//     PlcTask Inputs/MAIN.force_rb_Y[62] <-> Status process data mapping/force_rb_Y
//     PlcTask Inputs/MAIN.force_rb_Z[62] <-> Status process data mapping/force_rb_Z
//     PlcTask Inputs/MAIN.force_sp_X[62] <-> Status process data mapping/force_sp_X
//     PlcTask Inputs/MAIN.force_sp_Y[62] <-> Status process data mapping/force_sp_Y
//     PlcTask Inputs/MAIN.force_sp_Z[62] <-> Status process data mapping/force_sp_Z
//     PlcTask Inputs/MAIN.pwm1[62] <-> Status process data mapping/pwm1
//     PlcTask Inputs/MAIN.pwm2[62] <-> Status process data mapping/pwm2
//     PlcTask Inputs/MAIN.pwm3[62] <-> Status process data mapping/pwm3
//     PlcTask Outputs/MAIN.enable_cmd[62] <-> Control process data mapping/enable
//     PlcTask Outputs/MAIN.force_cmd_X[62] <-> Control process data mapping/force_sp_X
//     PlcTask Outputs/MAIN.force_cmd_Y[62] <-> Control process data mapping/force_sp_Y
//     PlcTask Outputs/MAIN.force_cmd_Z[62] <-> Control process data mapping/force_sp_Z
//     PlcTask Outputs/MAIN.msthb[67] <-> Control process data mapping/msthb
//   SAsetGains/SAsetGains Instance <-> Device 1 (EtherCAT)/Box 63 (m1eph)/Box 68 (m1sa)
//     PlcTask Inputs/MAIN.cloop_stat[63] <-> Status process data mapping/close_loop
//     PlcTask Inputs/MAIN.enable_stat[63] <-> Status process data mapping/enable
//     PlcTask Inputs/MAIN.force_rb_X[63] <-> Status process data mapping/force_rb_X
//     PlcTask Inputs/MAIN.force_rb_Y[63] <-> Status process data mapping/force_rb_Y
//     PlcTask Inputs/MAIN.force_rb_Z[63] <-> Status process data mapping/force_rb_Z
//     PlcTask Inputs/MAIN.force_sp_X[63] <-> Status process data mapping/force_sp_X
//     PlcTask Inputs/MAIN.force_sp_Y[63] <-> Status process data mapping/force_sp_Y
//     PlcTask Inputs/MAIN.force_sp_Z[63] <-> Status process data mapping/force_sp_Z
//     PlcTask Inputs/MAIN.pwm1[63] <-> Status process data mapping/pwm1
//     PlcTask Inputs/MAIN.pwm2[63] <-> Status process data mapping/pwm2
//     PlcTask Inputs/MAIN.pwm3[63] <-> Status process data mapping/pwm3
//     PlcTask Outputs/MAIN.enable_cmd[63] <-> Control process data mapping/enable
//     PlcTask Outputs/MAIN.force_cmd_X[63] <-> Control process data mapping/force_sp_X
//     PlcTask Outputs/MAIN.force_cmd_Y[63] <-> Control process data mapping/force_sp_Y
//     PlcTask Outputs/MAIN.force_cmd_Z[63] <-> Control process data mapping/force_sp_Z
//     PlcTask Outputs/MAIN.msthb[68] <-> Control process data mapping/msthb
//   SAsetGains/SAsetGains Instance <-> Device 1 (EtherCAT)/Box 63 (m1eph)/Box 69 (m1sa)
//     PlcTask Inputs/MAIN.cloop_stat[64] <-> Status process data mapping/close_loop
//     PlcTask Inputs/MAIN.enable_stat[64] <-> Status process data mapping/enable
//     PlcTask Inputs/MAIN.force_rb_X[64] <-> Status process data mapping/force_rb_X
//     PlcTask Inputs/MAIN.force_rb_Y[64] <-> Status process data mapping/force_rb_Y
//     PlcTask Inputs/MAIN.force_rb_Z[64] <-> Status process data mapping/force_rb_Z
//     PlcTask Inputs/MAIN.force_sp_X[64] <-> Status process data mapping/force_sp_X
//     PlcTask Inputs/MAIN.force_sp_Y[64] <-> Status process data mapping/force_sp_Y
//     PlcTask Inputs/MAIN.force_sp_Z[64] <-> Status process data mapping/force_sp_Z
//     PlcTask Inputs/MAIN.pwm1[64] <-> Status process data mapping/pwm1
//     PlcTask Inputs/MAIN.pwm2[64] <-> Status process data mapping/pwm2
//     PlcTask Inputs/MAIN.pwm3[64] <-> Status process data mapping/pwm3
//     PlcTask Outputs/MAIN.enable_cmd[64] <-> Control process data mapping/enable
//     PlcTask Outputs/MAIN.force_cmd_X[64] <-> Control process data mapping/force_sp_X
//     PlcTask Outputs/MAIN.force_cmd_Y[64] <-> Control process data mapping/force_sp_Y
//     PlcTask Outputs/MAIN.force_cmd_Z[64] <-> Control process data mapping/force_sp_Z
//     PlcTask Outputs/MAIN.msthb[69] <-> Control process data mapping/msthb
//   SAsetGains/SAsetGains Instance <-> Device 1 (EtherCAT)/Box 63 (m1eph)/Box 70 (m1sa)
//     PlcTask Inputs/MAIN.cloop_stat[65] <-> Status process data mapping/close_loop
//     PlcTask Inputs/MAIN.enable_stat[65] <-> Status process data mapping/enable
//     PlcTask Inputs/MAIN.force_rb_X[65] <-> Status process data mapping/force_rb_X
//     PlcTask Inputs/MAIN.force_rb_Y[65] <-> Status process data mapping/force_rb_Y
//     PlcTask Inputs/MAIN.force_rb_Z[65] <-> Status process data mapping/force_rb_Z
//     PlcTask Inputs/MAIN.force_sp_X[65] <-> Status process data mapping/force_sp_X
//     PlcTask Inputs/MAIN.force_sp_Y[65] <-> Status process data mapping/force_sp_Y
//     PlcTask Inputs/MAIN.force_sp_Z[65] <-> Status process data mapping/force_sp_Z
//     PlcTask Inputs/MAIN.pwm1[65] <-> Status process data mapping/pwm1
//     PlcTask Inputs/MAIN.pwm2[65] <-> Status process data mapping/pwm2
//     PlcTask Inputs/MAIN.pwm3[65] <-> Status process data mapping/pwm3
//     PlcTask Outputs/MAIN.enable_cmd[65] <-> Control process data mapping/enable
//     PlcTask Outputs/MAIN.force_cmd_X[65] <-> Control process data mapping/force_sp_X
//     PlcTask Outputs/MAIN.force_cmd_Y[65] <-> Control process data mapping/force_sp_Y
//     PlcTask Outputs/MAIN.force_cmd_Z[65] <-> Control process data mapping/force_sp_Z
//     PlcTask Outputs/MAIN.msthb[70] <-> Control process data mapping/msthb
//   SAsetGains/SAsetGains Instance <-> Device 1 (EtherCAT)/Box 63 (m1eph)/Box 71 (m1sa)
//     PlcTask Inputs/MAIN.cloop_stat[66] <-> Status process data mapping/close_loop
//     PlcTask Inputs/MAIN.enable_stat[66] <-> Status process data mapping/enable
//     PlcTask Inputs/MAIN.force_rb_X[66] <-> Status process data mapping/force_rb_X
//     PlcTask Inputs/MAIN.force_rb_Y[66] <-> Status process data mapping/force_rb_Y
//     PlcTask Inputs/MAIN.force_rb_Z[66] <-> Status process data mapping/force_rb_Z
//     PlcTask Inputs/MAIN.force_sp_X[66] <-> Status process data mapping/force_sp_X
//     PlcTask Inputs/MAIN.force_sp_Y[66] <-> Status process data mapping/force_sp_Y
//     PlcTask Inputs/MAIN.force_sp_Z[66] <-> Status process data mapping/force_sp_Z
//     PlcTask Inputs/MAIN.pwm1[66] <-> Status process data mapping/pwm1
//     PlcTask Inputs/MAIN.pwm2[66] <-> Status process data mapping/pwm2
//     PlcTask Inputs/MAIN.pwm3[66] <-> Status process data mapping/pwm3
//     PlcTask Outputs/MAIN.enable_cmd[66] <-> Control process data mapping/enable
//     PlcTask Outputs/MAIN.force_cmd_X[66] <-> Control process data mapping/force_sp_X
//     PlcTask Outputs/MAIN.force_cmd_Y[66] <-> Control process data mapping/force_sp_Y
//     PlcTask Outputs/MAIN.force_cmd_Z[66] <-> Control process data mapping/force_sp_Z
//     PlcTask Outputs/MAIN.msthb[71] <-> Control process data mapping/msthb
//   SAsetGains/SAsetGains Instance <-> Device 1 (EtherCAT)/Box 63 (m1eph)/Box 72 (m1sa)
//     PlcTask Inputs/MAIN.cloop_stat[67] <-> Status process data mapping/close_loop
//     PlcTask Inputs/MAIN.enable_stat[67] <-> Status process data mapping/enable
//     PlcTask Inputs/MAIN.force_rb_X[67] <-> Status process data mapping/force_rb_X
//     PlcTask Inputs/MAIN.force_rb_Y[67] <-> Status process data mapping/force_rb_Y
//     PlcTask Inputs/MAIN.force_rb_Z[67] <-> Status process data mapping/force_rb_Z
//     PlcTask Inputs/MAIN.force_sp_X[67] <-> Status process data mapping/force_sp_X
//     PlcTask Inputs/MAIN.force_sp_Y[67] <-> Status process data mapping/force_sp_Y
//     PlcTask Inputs/MAIN.force_sp_Z[67] <-> Status process data mapping/force_sp_Z
//     PlcTask Inputs/MAIN.pwm1[67] <-> Status process data mapping/pwm1
//     PlcTask Inputs/MAIN.pwm2[67] <-> Status process data mapping/pwm2
//     PlcTask Inputs/MAIN.pwm3[67] <-> Status process data mapping/pwm3
//     PlcTask Outputs/MAIN.enable_cmd[67] <-> Control process data mapping/enable
//     PlcTask Outputs/MAIN.force_cmd_X[67] <-> Control process data mapping/force_sp_X
//     PlcTask Outputs/MAIN.force_cmd_Y[67] <-> Control process data mapping/force_sp_Y
//     PlcTask Outputs/MAIN.force_cmd_Z[67] <-> Control process data mapping/force_sp_Z
//     PlcTask Outputs/MAIN.msthb[72] <-> Control process data mapping/msthb
//   SAsetGains/SAsetGains Instance <-> Device 1 (EtherCAT)/Box 63 (m1eph)/Box 73 (m1sa)
//     PlcTask Inputs/MAIN.cloop_stat[68] <-> Status process data mapping/close_loop
//     PlcTask Inputs/MAIN.enable_stat[68] <-> Status process data mapping/enable
//     PlcTask Inputs/MAIN.force_rb_X[68] <-> Status process data mapping/force_rb_X
//     PlcTask Inputs/MAIN.force_rb_Y[68] <-> Status process data mapping/force_rb_Y
//     PlcTask Inputs/MAIN.force_rb_Z[68] <-> Status process data mapping/force_rb_Z
//     PlcTask Inputs/MAIN.force_sp_X[68] <-> Status process data mapping/force_sp_X
//     PlcTask Inputs/MAIN.force_sp_Y[68] <-> Status process data mapping/force_sp_Y
//     PlcTask Inputs/MAIN.force_sp_Z[68] <-> Status process data mapping/force_sp_Z
//     PlcTask Inputs/MAIN.pwm1[68] <-> Status process data mapping/pwm1
//     PlcTask Inputs/MAIN.pwm2[68] <-> Status process data mapping/pwm2
//     PlcTask Inputs/MAIN.pwm3[68] <-> Status process data mapping/pwm3
//     PlcTask Outputs/MAIN.enable_cmd[68] <-> Control process data mapping/enable
//     PlcTask Outputs/MAIN.force_cmd_X[68] <-> Control process data mapping/force_sp_X
//     PlcTask Outputs/MAIN.force_cmd_Y[68] <-> Control process data mapping/force_sp_Y
//     PlcTask Outputs/MAIN.force_cmd_Z[68] <-> Control process data mapping/force_sp_Z
//     PlcTask Outputs/MAIN.msthb[73] <-> Control process data mapping/msthb
//   SAsetGains/SAsetGains Instance <-> Device 1 (EtherCAT)/Box 63 (m1eph)/Box 74 (m1sa)
//     PlcTask Inputs/MAIN.cloop_stat[69] <-> Status process data mapping/close_loop
//     PlcTask Inputs/MAIN.enable_stat[69] <-> Status process data mapping/enable
//     PlcTask Inputs/MAIN.force_rb_X[69] <-> Status process data mapping/force_rb_X
//     PlcTask Inputs/MAIN.force_rb_Y[69] <-> Status process data mapping/force_rb_Y
//     PlcTask Inputs/MAIN.force_rb_Z[69] <-> Status process data mapping/force_rb_Z
//     PlcTask Inputs/MAIN.force_sp_X[69] <-> Status process data mapping/force_sp_X
//     PlcTask Inputs/MAIN.force_sp_Y[69] <-> Status process data mapping/force_sp_Y
//     PlcTask Inputs/MAIN.force_sp_Z[69] <-> Status process data mapping/force_sp_Z
//     PlcTask Inputs/MAIN.pwm1[69] <-> Status process data mapping/pwm1
//     PlcTask Inputs/MAIN.pwm2[69] <-> Status process data mapping/pwm2
//     PlcTask Inputs/MAIN.pwm3[69] <-> Status process data mapping/pwm3
//     PlcTask Outputs/MAIN.enable_cmd[69] <-> Control process data mapping/enable
//     PlcTask Outputs/MAIN.force_cmd_X[69] <-> Control process data mapping/force_sp_X
//     PlcTask Outputs/MAIN.force_cmd_Y[69] <-> Control process data mapping/force_sp_Y
//     PlcTask Outputs/MAIN.force_cmd_Z[69] <-> Control process data mapping/force_sp_Z
//     PlcTask Outputs/MAIN.msthb[74] <-> Control process data mapping/msthb
//   SAsetGains/SAsetGains Instance <-> Device 1 (EtherCAT)/Box 63 (m1eph)/Box 75 (m1sa)
//     PlcTask Inputs/MAIN.cloop_stat[70] <-> Status process data mapping/close_loop
//     PlcTask Inputs/MAIN.enable_stat[70] <-> Status process data mapping/enable
//     PlcTask Inputs/MAIN.force_rb_X[70] <-> Status process data mapping/force_rb_X
//     PlcTask Inputs/MAIN.force_rb_Y[70] <-> Status process data mapping/force_rb_Y
//     PlcTask Inputs/MAIN.force_rb_Z[70] <-> Status process data mapping/force_rb_Z
//     PlcTask Inputs/MAIN.force_sp_X[70] <-> Status process data mapping/force_sp_X
//     PlcTask Inputs/MAIN.force_sp_Y[70] <-> Status process data mapping/force_sp_Y
//     PlcTask Inputs/MAIN.force_sp_Z[70] <-> Status process data mapping/force_sp_Z
//     PlcTask Inputs/MAIN.pwm1[70] <-> Status process data mapping/pwm1
//     PlcTask Inputs/MAIN.pwm2[70] <-> Status process data mapping/pwm2
//     PlcTask Inputs/MAIN.pwm3[70] <-> Status process data mapping/pwm3
//     PlcTask Outputs/MAIN.enable_cmd[70] <-> Control process data mapping/enable
//     PlcTask Outputs/MAIN.force_cmd_X[70] <-> Control process data mapping/force_sp_X
//     PlcTask Outputs/MAIN.force_cmd_Y[70] <-> Control process data mapping/force_sp_Y
//     PlcTask Outputs/MAIN.force_cmd_Z[70] <-> Control process data mapping/force_sp_Z
//     PlcTask Outputs/MAIN.msthb[75] <-> Control process data mapping/msthb
//   SAsetGains/SAsetGains Instance <-> Device 1 (EtherCAT)/Box 63 (m1eph)/Box 76 (m1sa)
//     PlcTask Inputs/MAIN.cloop_stat[71] <-> Status process data mapping/close_loop
//     PlcTask Inputs/MAIN.enable_stat[71] <-> Status process data mapping/enable
//     PlcTask Inputs/MAIN.force_rb_X[71] <-> Status process data mapping/force_rb_X
//     PlcTask Inputs/MAIN.force_rb_Y[71] <-> Status process data mapping/force_rb_Y
//     PlcTask Inputs/MAIN.force_rb_Z[71] <-> Status process data mapping/force_rb_Z
//     PlcTask Inputs/MAIN.force_sp_X[71] <-> Status process data mapping/force_sp_X
//     PlcTask Inputs/MAIN.force_sp_Y[71] <-> Status process data mapping/force_sp_Y
//     PlcTask Inputs/MAIN.force_sp_Z[71] <-> Status process data mapping/force_sp_Z
//     PlcTask Inputs/MAIN.pwm1[71] <-> Status process data mapping/pwm1
//     PlcTask Inputs/MAIN.pwm2[71] <-> Status process data mapping/pwm2
//     PlcTask Inputs/MAIN.pwm3[71] <-> Status process data mapping/pwm3
//     PlcTask Outputs/MAIN.enable_cmd[71] <-> Control process data mapping/enable
//     PlcTask Outputs/MAIN.force_cmd_X[71] <-> Control process data mapping/force_sp_X
//     PlcTask Outputs/MAIN.force_cmd_Y[71] <-> Control process data mapping/force_sp_Y
//     PlcTask Outputs/MAIN.force_cmd_Z[71] <-> Control process data mapping/force_sp_Z
//     PlcTask Outputs/MAIN.msthb[76] <-> Control process data mapping/msthb
//   SAsetGains/SAsetGains Instance <-> Device 1 (EtherCAT)/Box 63 (m1eph)/Box 77 (m1sa)
//     PlcTask Inputs/MAIN.cloop_stat[72] <-> Status process data mapping/close_loop
//     PlcTask Inputs/MAIN.enable_stat[72] <-> Status process data mapping/enable
//     PlcTask Inputs/MAIN.force_rb_X[72] <-> Status process data mapping/force_rb_X
//     PlcTask Inputs/MAIN.force_rb_Y[72] <-> Status process data mapping/force_rb_Y
//     PlcTask Inputs/MAIN.force_rb_Z[72] <-> Status process data mapping/force_rb_Z
//     PlcTask Inputs/MAIN.force_sp_X[72] <-> Status process data mapping/force_sp_X
//     PlcTask Inputs/MAIN.force_sp_Y[72] <-> Status process data mapping/force_sp_Y
//     PlcTask Inputs/MAIN.force_sp_Z[72] <-> Status process data mapping/force_sp_Z
//     PlcTask Inputs/MAIN.pwm1[72] <-> Status process data mapping/pwm1
//     PlcTask Inputs/MAIN.pwm2[72] <-> Status process data mapping/pwm2
//     PlcTask Inputs/MAIN.pwm3[72] <-> Status process data mapping/pwm3
//     PlcTask Outputs/MAIN.enable_cmd[72] <-> Control process data mapping/enable
//     PlcTask Outputs/MAIN.force_cmd_X[72] <-> Control process data mapping/force_sp_X
//     PlcTask Outputs/MAIN.force_cmd_Y[72] <-> Control process data mapping/force_sp_Y
//     PlcTask Outputs/MAIN.force_cmd_Z[72] <-> Control process data mapping/force_sp_Z
//     PlcTask Outputs/MAIN.msthb[77] <-> Control process data mapping/msthb
//   SAsetGains/SAsetGains Instance <-> Device 1 (EtherCAT)/Box 63 (m1eph)/Box 78 (m1sa)
//     PlcTask Inputs/MAIN.cloop_stat[73] <-> Status process data mapping/close_loop
//     PlcTask Inputs/MAIN.enable_stat[73] <-> Status process data mapping/enable
//     PlcTask Inputs/MAIN.force_rb_X[73] <-> Status process data mapping/force_rb_X
//     PlcTask Inputs/MAIN.force_rb_Y[73] <-> Status process data mapping/force_rb_Y
//     PlcTask Inputs/MAIN.force_rb_Z[73] <-> Status process data mapping/force_rb_Z
//     PlcTask Inputs/MAIN.force_sp_X[73] <-> Status process data mapping/force_sp_X
//     PlcTask Inputs/MAIN.force_sp_Y[73] <-> Status process data mapping/force_sp_Y
//     PlcTask Inputs/MAIN.force_sp_Z[73] <-> Status process data mapping/force_sp_Z
//     PlcTask Inputs/MAIN.pwm1[73] <-> Status process data mapping/pwm1
//     PlcTask Inputs/MAIN.pwm2[73] <-> Status process data mapping/pwm2
//     PlcTask Inputs/MAIN.pwm3[73] <-> Status process data mapping/pwm3
//     PlcTask Outputs/MAIN.enable_cmd[73] <-> Control process data mapping/enable
//     PlcTask Outputs/MAIN.force_cmd_X[73] <-> Control process data mapping/force_sp_X
//     PlcTask Outputs/MAIN.force_cmd_Y[73] <-> Control process data mapping/force_sp_Y
//     PlcTask Outputs/MAIN.force_cmd_Z[73] <-> Control process data mapping/force_sp_Z
//     PlcTask Outputs/MAIN.msthb[78] <-> Control process data mapping/msthb
//   SAsetGains/SAsetGains Instance <-> Device 1 (EtherCAT)/Box 63 (m1eph)/Box 79 (m1sa)
//     PlcTask Inputs/MAIN.cloop_stat[74] <-> Status process data mapping/close_loop
//     PlcTask Inputs/MAIN.enable_stat[74] <-> Status process data mapping/enable
//     PlcTask Inputs/MAIN.force_rb_X[74] <-> Status process data mapping/force_rb_X
//     PlcTask Inputs/MAIN.force_rb_Y[74] <-> Status process data mapping/force_rb_Y
//     PlcTask Inputs/MAIN.force_rb_Z[74] <-> Status process data mapping/force_rb_Z
//     PlcTask Inputs/MAIN.force_sp_X[74] <-> Status process data mapping/force_sp_X
//     PlcTask Inputs/MAIN.force_sp_Y[74] <-> Status process data mapping/force_sp_Y
//     PlcTask Inputs/MAIN.force_sp_Z[74] <-> Status process data mapping/force_sp_Z
//     PlcTask Inputs/MAIN.pwm1[74] <-> Status process data mapping/pwm1
//     PlcTask Inputs/MAIN.pwm2[74] <-> Status process data mapping/pwm2
//     PlcTask Inputs/MAIN.pwm3[74] <-> Status process data mapping/pwm3
//     PlcTask Outputs/MAIN.enable_cmd[74] <-> Control process data mapping/enable
//     PlcTask Outputs/MAIN.force_cmd_X[74] <-> Control process data mapping/force_sp_X
//     PlcTask Outputs/MAIN.force_cmd_Y[74] <-> Control process data mapping/force_sp_Y
//     PlcTask Outputs/MAIN.force_cmd_Z[74] <-> Control process data mapping/force_sp_Z
//     PlcTask Outputs/MAIN.msthb[79] <-> Control process data mapping/msthb
//   SAsetGains/SAsetGains Instance <-> Device 1 (EtherCAT)/Box 80 (m1eph)
//     PlcTask Outputs/MAIN.msthb[80] <-> Control process data mapping/msthb
//   SAsetGains/SAsetGains Instance <-> Device 1 (EtherCAT)/Box 80 (m1eph)/Box 81 (m1sa)
//     PlcTask Inputs/MAIN.cloop_stat[75] <-> Status process data mapping/close_loop
//     PlcTask Inputs/MAIN.enable_stat[75] <-> Status process data mapping/enable
//     PlcTask Inputs/MAIN.force_rb_X[75] <-> Status process data mapping/force_rb_X
//     PlcTask Inputs/MAIN.force_rb_Y[75] <-> Status process data mapping/force_rb_Y
//     PlcTask Inputs/MAIN.force_rb_Z[75] <-> Status process data mapping/force_rb_Z
//     PlcTask Inputs/MAIN.force_sp_X[75] <-> Status process data mapping/force_sp_X
//     PlcTask Inputs/MAIN.force_sp_Y[75] <-> Status process data mapping/force_sp_Y
//     PlcTask Inputs/MAIN.force_sp_Z[75] <-> Status process data mapping/force_sp_Z
//     PlcTask Inputs/MAIN.pwm1[75] <-> Status process data mapping/pwm1
//     PlcTask Inputs/MAIN.pwm2[75] <-> Status process data mapping/pwm2
//     PlcTask Inputs/MAIN.pwm3[75] <-> Status process data mapping/pwm3
//     PlcTask Outputs/MAIN.enable_cmd[75] <-> Control process data mapping/enable
//     PlcTask Outputs/MAIN.force_cmd_X[75] <-> Control process data mapping/force_sp_X
//     PlcTask Outputs/MAIN.force_cmd_Y[75] <-> Control process data mapping/force_sp_Y
//     PlcTask Outputs/MAIN.force_cmd_Z[75] <-> Control process data mapping/force_sp_Z
//     PlcTask Outputs/MAIN.msthb[81] <-> Control process data mapping/msthb
//   SAsetGains/SAsetGains Instance <-> Device 1 (EtherCAT)/Box 80 (m1eph)/Box 82 (m1sa)
//     PlcTask Inputs/MAIN.cloop_stat[76] <-> Status process data mapping/close_loop
//     PlcTask Inputs/MAIN.enable_stat[76] <-> Status process data mapping/enable
//     PlcTask Inputs/MAIN.force_rb_X[76] <-> Status process data mapping/force_rb_X
//     PlcTask Inputs/MAIN.force_rb_Y[76] <-> Status process data mapping/force_rb_Y
//     PlcTask Inputs/MAIN.force_rb_Z[76] <-> Status process data mapping/force_rb_Z
//     PlcTask Inputs/MAIN.force_sp_X[76] <-> Status process data mapping/force_sp_X
//     PlcTask Inputs/MAIN.force_sp_Y[76] <-> Status process data mapping/force_sp_Y
//     PlcTask Inputs/MAIN.force_sp_Z[76] <-> Status process data mapping/force_sp_Z
//     PlcTask Inputs/MAIN.pwm1[76] <-> Status process data mapping/pwm1
//     PlcTask Inputs/MAIN.pwm2[76] <-> Status process data mapping/pwm2
//     PlcTask Inputs/MAIN.pwm3[76] <-> Status process data mapping/pwm3
//     PlcTask Outputs/MAIN.enable_cmd[76] <-> Control process data mapping/enable
//     PlcTask Outputs/MAIN.force_cmd_X[76] <-> Control process data mapping/force_sp_X
//     PlcTask Outputs/MAIN.force_cmd_Y[76] <-> Control process data mapping/force_sp_Y
//     PlcTask Outputs/MAIN.force_cmd_Z[76] <-> Control process data mapping/force_sp_Z
//     PlcTask Outputs/MAIN.msthb[82] <-> Control process data mapping/msthb
//   SAsetGains/SAsetGains Instance <-> Device 1 (EtherCAT)/Box 80 (m1eph)/Box 83 (m1sa)
//     PlcTask Inputs/MAIN.cloop_stat[77] <-> Status process data mapping/close_loop
//     PlcTask Inputs/MAIN.enable_stat[77] <-> Status process data mapping/enable
//     PlcTask Inputs/MAIN.force_rb_X[77] <-> Status process data mapping/force_rb_X
//     PlcTask Inputs/MAIN.force_rb_Y[77] <-> Status process data mapping/force_rb_Y
//     PlcTask Inputs/MAIN.force_rb_Z[77] <-> Status process data mapping/force_rb_Z
//     PlcTask Inputs/MAIN.force_sp_X[77] <-> Status process data mapping/force_sp_X
//     PlcTask Inputs/MAIN.force_sp_Y[77] <-> Status process data mapping/force_sp_Y
//     PlcTask Inputs/MAIN.force_sp_Z[77] <-> Status process data mapping/force_sp_Z
//     PlcTask Inputs/MAIN.pwm1[77] <-> Status process data mapping/pwm1
//     PlcTask Inputs/MAIN.pwm2[77] <-> Status process data mapping/pwm2
//     PlcTask Inputs/MAIN.pwm3[77] <-> Status process data mapping/pwm3
//     PlcTask Outputs/MAIN.enable_cmd[77] <-> Control process data mapping/enable
//     PlcTask Outputs/MAIN.force_cmd_X[77] <-> Control process data mapping/force_sp_X
//     PlcTask Outputs/MAIN.force_cmd_Y[77] <-> Control process data mapping/force_sp_Y
//     PlcTask Outputs/MAIN.force_cmd_Z[77] <-> Control process data mapping/force_sp_Z
//     PlcTask Outputs/MAIN.msthb[83] <-> Control process data mapping/msthb
//   SAsetGains/SAsetGains Instance <-> Device 1 (EtherCAT)/Box 80 (m1eph)/Box 84 (m1sa)
//     PlcTask Inputs/MAIN.cloop_stat[78] <-> Status process data mapping/close_loop
//     PlcTask Inputs/MAIN.enable_stat[78] <-> Status process data mapping/enable
//     PlcTask Inputs/MAIN.force_rb_X[78] <-> Status process data mapping/force_rb_X
//     PlcTask Inputs/MAIN.force_rb_Y[78] <-> Status process data mapping/force_rb_Y
//     PlcTask Inputs/MAIN.force_rb_Z[78] <-> Status process data mapping/force_rb_Z
//     PlcTask Inputs/MAIN.force_sp_X[78] <-> Status process data mapping/force_sp_X
//     PlcTask Inputs/MAIN.force_sp_Y[78] <-> Status process data mapping/force_sp_Y
//     PlcTask Inputs/MAIN.force_sp_Z[78] <-> Status process data mapping/force_sp_Z
//     PlcTask Inputs/MAIN.pwm1[78] <-> Status process data mapping/pwm1
//     PlcTask Inputs/MAIN.pwm2[78] <-> Status process data mapping/pwm2
//     PlcTask Inputs/MAIN.pwm3[78] <-> Status process data mapping/pwm3
//     PlcTask Outputs/MAIN.enable_cmd[78] <-> Control process data mapping/enable
//     PlcTask Outputs/MAIN.force_cmd_X[78] <-> Control process data mapping/force_sp_X
//     PlcTask Outputs/MAIN.force_cmd_Y[78] <-> Control process data mapping/force_sp_Y
//     PlcTask Outputs/MAIN.force_cmd_Z[78] <-> Control process data mapping/force_sp_Z
//     PlcTask Outputs/MAIN.msthb[84] <-> Control process data mapping/msthb
//   SAsetGains/SAsetGains Instance <-> Device 1 (EtherCAT)/Box 80 (m1eph)/Box 85 (m1sa)
//     PlcTask Inputs/MAIN.cloop_stat[79] <-> Status process data mapping/close_loop
//     PlcTask Inputs/MAIN.enable_stat[79] <-> Status process data mapping/enable
//     PlcTask Inputs/MAIN.force_rb_X[79] <-> Status process data mapping/force_rb_X
//     PlcTask Inputs/MAIN.force_rb_Y[79] <-> Status process data mapping/force_rb_Y
//     PlcTask Inputs/MAIN.force_rb_Z[79] <-> Status process data mapping/force_rb_Z
//     PlcTask Inputs/MAIN.force_sp_X[79] <-> Status process data mapping/force_sp_X
//     PlcTask Inputs/MAIN.force_sp_Y[79] <-> Status process data mapping/force_sp_Y
//     PlcTask Inputs/MAIN.force_sp_Z[79] <-> Status process data mapping/force_sp_Z
//     PlcTask Inputs/MAIN.pwm1[79] <-> Status process data mapping/pwm1
//     PlcTask Inputs/MAIN.pwm2[79] <-> Status process data mapping/pwm2
//     PlcTask Inputs/MAIN.pwm3[79] <-> Status process data mapping/pwm3
//     PlcTask Outputs/MAIN.enable_cmd[79] <-> Control process data mapping/enable
//     PlcTask Outputs/MAIN.force_cmd_X[79] <-> Control process data mapping/force_sp_X
//     PlcTask Outputs/MAIN.force_cmd_Y[79] <-> Control process data mapping/force_sp_Y
//     PlcTask Outputs/MAIN.force_cmd_Z[79] <-> Control process data mapping/force_sp_Z
//     PlcTask Outputs/MAIN.msthb[85] <-> Control process data mapping/msthb
//   SAsetGains/SAsetGains Instance <-> Device 1 (EtherCAT)/Box 80 (m1eph)/Box 86 (m1sa)
//     PlcTask Inputs/MAIN.cloop_stat[80] <-> Status process data mapping/close_loop
//     PlcTask Inputs/MAIN.enable_stat[80] <-> Status process data mapping/enable
//     PlcTask Inputs/MAIN.force_rb_X[80] <-> Status process data mapping/force_rb_X
//     PlcTask Inputs/MAIN.force_rb_Y[80] <-> Status process data mapping/force_rb_Y
//     PlcTask Inputs/MAIN.force_rb_Z[80] <-> Status process data mapping/force_rb_Z
//     PlcTask Inputs/MAIN.force_sp_X[80] <-> Status process data mapping/force_sp_X
//     PlcTask Inputs/MAIN.force_sp_Y[80] <-> Status process data mapping/force_sp_Y
//     PlcTask Inputs/MAIN.force_sp_Z[80] <-> Status process data mapping/force_sp_Z
//     PlcTask Inputs/MAIN.pwm1[80] <-> Status process data mapping/pwm1
//     PlcTask Inputs/MAIN.pwm2[80] <-> Status process data mapping/pwm2
//     PlcTask Inputs/MAIN.pwm3[80] <-> Status process data mapping/pwm3
//     PlcTask Outputs/MAIN.enable_cmd[80] <-> Control process data mapping/enable
//     PlcTask Outputs/MAIN.force_cmd_X[80] <-> Control process data mapping/force_sp_X
//     PlcTask Outputs/MAIN.force_cmd_Y[80] <-> Control process data mapping/force_sp_Y
//     PlcTask Outputs/MAIN.force_cmd_Z[80] <-> Control process data mapping/force_sp_Z
//     PlcTask Outputs/MAIN.msthb[86] <-> Control process data mapping/msthb
//   SAsetGains/SAsetGains Instance <-> Device 1 (EtherCAT)/Box 80 (m1eph)/Box 87 (m1sa)
//     PlcTask Inputs/MAIN.cloop_stat[81] <-> Status process data mapping/close_loop
//     PlcTask Inputs/MAIN.enable_stat[81] <-> Status process data mapping/enable
//     PlcTask Inputs/MAIN.force_rb_X[81] <-> Status process data mapping/force_rb_X
//     PlcTask Inputs/MAIN.force_rb_Y[81] <-> Status process data mapping/force_rb_Y
//     PlcTask Inputs/MAIN.force_rb_Z[81] <-> Status process data mapping/force_rb_Z
//     PlcTask Inputs/MAIN.force_sp_X[81] <-> Status process data mapping/force_sp_X
//     PlcTask Inputs/MAIN.force_sp_Y[81] <-> Status process data mapping/force_sp_Y
//     PlcTask Inputs/MAIN.force_sp_Z[81] <-> Status process data mapping/force_sp_Z
//     PlcTask Inputs/MAIN.pwm1[81] <-> Status process data mapping/pwm1
//     PlcTask Inputs/MAIN.pwm2[81] <-> Status process data mapping/pwm2
//     PlcTask Inputs/MAIN.pwm3[81] <-> Status process data mapping/pwm3
//     PlcTask Outputs/MAIN.enable_cmd[81] <-> Control process data mapping/enable
//     PlcTask Outputs/MAIN.force_cmd_X[81] <-> Control process data mapping/force_sp_X
//     PlcTask Outputs/MAIN.force_cmd_Y[81] <-> Control process data mapping/force_sp_Y
//     PlcTask Outputs/MAIN.force_cmd_Z[81] <-> Control process data mapping/force_sp_Z
//     PlcTask Outputs/MAIN.msthb[87] <-> Control process data mapping/msthb
//   SAsetGains/SAsetGains Instance <-> Device 1 (EtherCAT)/Box 80 (m1eph)/Box 88 (m1sa)
//     PlcTask Inputs/MAIN.cloop_stat[82] <-> Status process data mapping/close_loop
//     PlcTask Inputs/MAIN.enable_stat[82] <-> Status process data mapping/enable
//     PlcTask Inputs/MAIN.force_rb_X[82] <-> Status process data mapping/force_rb_X
//     PlcTask Inputs/MAIN.force_rb_Y[82] <-> Status process data mapping/force_rb_Y
//     PlcTask Inputs/MAIN.force_rb_Z[82] <-> Status process data mapping/force_rb_Z
//     PlcTask Inputs/MAIN.force_sp_X[82] <-> Status process data mapping/force_sp_X
//     PlcTask Inputs/MAIN.force_sp_Y[82] <-> Status process data mapping/force_sp_Y
//     PlcTask Inputs/MAIN.force_sp_Z[82] <-> Status process data mapping/force_sp_Z
//     PlcTask Inputs/MAIN.pwm1[82] <-> Status process data mapping/pwm1
//     PlcTask Inputs/MAIN.pwm2[82] <-> Status process data mapping/pwm2
//     PlcTask Inputs/MAIN.pwm3[82] <-> Status process data mapping/pwm3
//     PlcTask Outputs/MAIN.enable_cmd[82] <-> Control process data mapping/enable
//     PlcTask Outputs/MAIN.force_cmd_X[82] <-> Control process data mapping/force_sp_X
//     PlcTask Outputs/MAIN.force_cmd_Y[82] <-> Control process data mapping/force_sp_Y
//     PlcTask Outputs/MAIN.force_cmd_Z[82] <-> Control process data mapping/force_sp_Z
//     PlcTask Outputs/MAIN.msthb[88] <-> Control process data mapping/msthb
//   SAsetGains/SAsetGains Instance <-> Device 1 (EtherCAT)/Box 80 (m1eph)/Box 89 (m1sa)
//     PlcTask Inputs/MAIN.cloop_stat[83] <-> Status process data mapping/close_loop
//     PlcTask Inputs/MAIN.enable_stat[83] <-> Status process data mapping/enable
//     PlcTask Inputs/MAIN.force_rb_X[83] <-> Status process data mapping/force_rb_X
//     PlcTask Inputs/MAIN.force_rb_Y[83] <-> Status process data mapping/force_rb_Y
//     PlcTask Inputs/MAIN.force_rb_Z[83] <-> Status process data mapping/force_rb_Z
//     PlcTask Inputs/MAIN.force_sp_X[83] <-> Status process data mapping/force_sp_X
//     PlcTask Inputs/MAIN.force_sp_Y[83] <-> Status process data mapping/force_sp_Y
//     PlcTask Inputs/MAIN.force_sp_Z[83] <-> Status process data mapping/force_sp_Z
//     PlcTask Inputs/MAIN.pwm1[83] <-> Status process data mapping/pwm1
//     PlcTask Inputs/MAIN.pwm2[83] <-> Status process data mapping/pwm2
//     PlcTask Inputs/MAIN.pwm3[83] <-> Status process data mapping/pwm3
//     PlcTask Outputs/MAIN.enable_cmd[83] <-> Control process data mapping/enable
//     PlcTask Outputs/MAIN.force_cmd_X[83] <-> Control process data mapping/force_sp_X
//     PlcTask Outputs/MAIN.force_cmd_Y[83] <-> Control process data mapping/force_sp_Y
//     PlcTask Outputs/MAIN.force_cmd_Z[83] <-> Control process data mapping/force_sp_Z
//     PlcTask Outputs/MAIN.msthb[89] <-> Control process data mapping/msthb
//   SAsetGains/SAsetGains Instance <-> Device 1 (EtherCAT)/Box 80 (m1eph)/Box 90 (m1sa)
//     PlcTask Inputs/MAIN.cloop_stat[84] <-> Status process data mapping/close_loop
//     PlcTask Inputs/MAIN.enable_stat[84] <-> Status process data mapping/enable
//     PlcTask Inputs/MAIN.force_rb_X[84] <-> Status process data mapping/force_rb_X
//     PlcTask Inputs/MAIN.force_rb_Y[84] <-> Status process data mapping/force_rb_Y
//     PlcTask Inputs/MAIN.force_rb_Z[84] <-> Status process data mapping/force_rb_Z
//     PlcTask Inputs/MAIN.force_sp_X[84] <-> Status process data mapping/force_sp_X
//     PlcTask Inputs/MAIN.force_sp_Y[84] <-> Status process data mapping/force_sp_Y
//     PlcTask Inputs/MAIN.force_sp_Z[84] <-> Status process data mapping/force_sp_Z
//     PlcTask Inputs/MAIN.pwm1[84] <-> Status process data mapping/pwm1
//     PlcTask Inputs/MAIN.pwm2[84] <-> Status process data mapping/pwm2
//     PlcTask Inputs/MAIN.pwm3[84] <-> Status process data mapping/pwm3
//     PlcTask Outputs/MAIN.enable_cmd[84] <-> Control process data mapping/enable
//     PlcTask Outputs/MAIN.force_cmd_X[84] <-> Control process data mapping/force_sp_X
//     PlcTask Outputs/MAIN.force_cmd_Y[84] <-> Control process data mapping/force_sp_Y
//     PlcTask Outputs/MAIN.force_cmd_Z[84] <-> Control process data mapping/force_sp_Z
//     PlcTask Outputs/MAIN.msthb[90] <-> Control process data mapping/msthb
//   SAsetGains/SAsetGains Instance <-> Device 1 (EtherCAT)/Box 80 (m1eph)/Box 91 (m1sa)
//     PlcTask Inputs/MAIN.cloop_stat[85] <-> Status process data mapping/close_loop
//     PlcTask Inputs/MAIN.enable_stat[85] <-> Status process data mapping/enable
//     PlcTask Inputs/MAIN.force_rb_X[85] <-> Status process data mapping/force_rb_X
//     PlcTask Inputs/MAIN.force_rb_Y[85] <-> Status process data mapping/force_rb_Y
//     PlcTask Inputs/MAIN.force_rb_Z[85] <-> Status process data mapping/force_rb_Z
//     PlcTask Inputs/MAIN.force_sp_X[85] <-> Status process data mapping/force_sp_X
//     PlcTask Inputs/MAIN.force_sp_Y[85] <-> Status process data mapping/force_sp_Y
//     PlcTask Inputs/MAIN.force_sp_Z[85] <-> Status process data mapping/force_sp_Z
//     PlcTask Inputs/MAIN.pwm1[85] <-> Status process data mapping/pwm1
//     PlcTask Inputs/MAIN.pwm2[85] <-> Status process data mapping/pwm2
//     PlcTask Inputs/MAIN.pwm3[85] <-> Status process data mapping/pwm3
//     PlcTask Outputs/MAIN.enable_cmd[85] <-> Control process data mapping/enable
//     PlcTask Outputs/MAIN.force_cmd_X[85] <-> Control process data mapping/force_sp_X
//     PlcTask Outputs/MAIN.force_cmd_Y[85] <-> Control process data mapping/force_sp_Y
//     PlcTask Outputs/MAIN.force_cmd_Z[85] <-> Control process data mapping/force_sp_Z
//     PlcTask Outputs/MAIN.msthb[91] <-> Control process data mapping/msthb
//   SAsetGains/SAsetGains Instance <-> Device 1 (EtherCAT)/Box 80 (m1eph)/Box 92 (m1sa)
//     PlcTask Inputs/MAIN.cloop_stat[86] <-> Status process data mapping/close_loop
//     PlcTask Inputs/MAIN.enable_stat[86] <-> Status process data mapping/enable
//     PlcTask Inputs/MAIN.force_rb_X[86] <-> Status process data mapping/force_rb_X
//     PlcTask Inputs/MAIN.force_rb_Y[86] <-> Status process data mapping/force_rb_Y
//     PlcTask Inputs/MAIN.force_rb_Z[86] <-> Status process data mapping/force_rb_Z
//     PlcTask Inputs/MAIN.force_sp_X[86] <-> Status process data mapping/force_sp_X
//     PlcTask Inputs/MAIN.force_sp_Y[86] <-> Status process data mapping/force_sp_Y
//     PlcTask Inputs/MAIN.force_sp_Z[86] <-> Status process data mapping/force_sp_Z
//     PlcTask Inputs/MAIN.pwm1[86] <-> Status process data mapping/pwm1
//     PlcTask Inputs/MAIN.pwm2[86] <-> Status process data mapping/pwm2
//     PlcTask Inputs/MAIN.pwm3[86] <-> Status process data mapping/pwm3
//     PlcTask Outputs/MAIN.enable_cmd[86] <-> Control process data mapping/enable
//     PlcTask Outputs/MAIN.force_cmd_X[86] <-> Control process data mapping/force_sp_X
//     PlcTask Outputs/MAIN.force_cmd_Y[86] <-> Control process data mapping/force_sp_Y
//     PlcTask Outputs/MAIN.force_cmd_Z[86] <-> Control process data mapping/force_sp_Z
//     PlcTask Outputs/MAIN.msthb[92] <-> Control process data mapping/msthb
//   SAsetGains/SAsetGains Instance <-> Device 1 (EtherCAT)/Box 80 (m1eph)/Box 93 (m1sa)
//     PlcTask Inputs/MAIN.cloop_stat[87] <-> Status process data mapping/close_loop
//     PlcTask Inputs/MAIN.enable_stat[87] <-> Status process data mapping/enable
//     PlcTask Inputs/MAIN.force_rb_X[87] <-> Status process data mapping/force_rb_X
//     PlcTask Inputs/MAIN.force_rb_Y[87] <-> Status process data mapping/force_rb_Y
//     PlcTask Inputs/MAIN.force_rb_Z[87] <-> Status process data mapping/force_rb_Z
//     PlcTask Inputs/MAIN.force_sp_X[87] <-> Status process data mapping/force_sp_X
//     PlcTask Inputs/MAIN.force_sp_Y[87] <-> Status process data mapping/force_sp_Y
//     PlcTask Inputs/MAIN.force_sp_Z[87] <-> Status process data mapping/force_sp_Z
//     PlcTask Inputs/MAIN.pwm1[87] <-> Status process data mapping/pwm1
//     PlcTask Inputs/MAIN.pwm2[87] <-> Status process data mapping/pwm2
//     PlcTask Inputs/MAIN.pwm3[87] <-> Status process data mapping/pwm3
//     PlcTask Outputs/MAIN.enable_cmd[87] <-> Control process data mapping/enable
//     PlcTask Outputs/MAIN.force_cmd_X[87] <-> Control process data mapping/force_sp_X
//     PlcTask Outputs/MAIN.force_cmd_Y[87] <-> Control process data mapping/force_sp_Y
//     PlcTask Outputs/MAIN.force_cmd_Z[87] <-> Control process data mapping/force_sp_Z
//     PlcTask Outputs/MAIN.msthb[93] <-> Control process data mapping/msthb
//   SAsetGains/SAsetGains Instance <-> Device 1 (EtherCAT)/Box 80 (m1eph)/Box 94 (m1sa)
//     PlcTask Inputs/MAIN.cloop_stat[88] <-> Status process data mapping/close_loop
//     PlcTask Inputs/MAIN.enable_stat[88] <-> Status process data mapping/enable
//     PlcTask Inputs/MAIN.force_rb_X[88] <-> Status process data mapping/force_rb_X
//     PlcTask Inputs/MAIN.force_rb_Y[88] <-> Status process data mapping/force_rb_Y
//     PlcTask Inputs/MAIN.force_rb_Z[88] <-> Status process data mapping/force_rb_Z
//     PlcTask Inputs/MAIN.force_sp_X[88] <-> Status process data mapping/force_sp_X
//     PlcTask Inputs/MAIN.force_sp_Y[88] <-> Status process data mapping/force_sp_Y
//     PlcTask Inputs/MAIN.force_sp_Z[88] <-> Status process data mapping/force_sp_Z
//     PlcTask Inputs/MAIN.pwm1[88] <-> Status process data mapping/pwm1
//     PlcTask Inputs/MAIN.pwm2[88] <-> Status process data mapping/pwm2
//     PlcTask Inputs/MAIN.pwm3[88] <-> Status process data mapping/pwm3
//     PlcTask Outputs/MAIN.enable_cmd[88] <-> Control process data mapping/enable
//     PlcTask Outputs/MAIN.force_cmd_X[88] <-> Control process data mapping/force_sp_X
//     PlcTask Outputs/MAIN.force_cmd_Y[88] <-> Control process data mapping/force_sp_Y
//     PlcTask Outputs/MAIN.force_cmd_Z[88] <-> Control process data mapping/force_sp_Z
//     PlcTask Outputs/MAIN.msthb[94] <-> Control process data mapping/msthb
//   SAsetGains/SAsetGains Instance <-> Device 1 (EtherCAT)/Box 80 (m1eph)/Box 95 (m1sa)
//     PlcTask Inputs/MAIN.cloop_stat[89] <-> Status process data mapping/close_loop
//     PlcTask Inputs/MAIN.enable_stat[89] <-> Status process data mapping/enable
//     PlcTask Inputs/MAIN.force_rb_X[89] <-> Status process data mapping/force_rb_X
//     PlcTask Inputs/MAIN.force_rb_Y[89] <-> Status process data mapping/force_rb_Y
//     PlcTask Inputs/MAIN.force_rb_Z[89] <-> Status process data mapping/force_rb_Z
//     PlcTask Inputs/MAIN.force_sp_X[89] <-> Status process data mapping/force_sp_X
//     PlcTask Inputs/MAIN.force_sp_Y[89] <-> Status process data mapping/force_sp_Y
//     PlcTask Inputs/MAIN.force_sp_Z[89] <-> Status process data mapping/force_sp_Z
//     PlcTask Inputs/MAIN.pwm1[89] <-> Status process data mapping/pwm1
//     PlcTask Inputs/MAIN.pwm2[89] <-> Status process data mapping/pwm2
//     PlcTask Inputs/MAIN.pwm3[89] <-> Status process data mapping/pwm3
//     PlcTask Outputs/MAIN.enable_cmd[89] <-> Control process data mapping/enable
//     PlcTask Outputs/MAIN.force_cmd_X[89] <-> Control process data mapping/force_sp_X
//     PlcTask Outputs/MAIN.force_cmd_Y[89] <-> Control process data mapping/force_sp_Y
//     PlcTask Outputs/MAIN.force_cmd_Z[89] <-> Control process data mapping/force_sp_Z
//     PlcTask Outputs/MAIN.msthb[95] <-> Control process data mapping/msthb
//   SAsetGains/SAsetGains Instance <-> Device 1 (EtherCAT)/Box 80 (m1eph)/Box 96 (m1sa)
//     PlcTask Inputs/MAIN.cloop_stat[90] <-> Status process data mapping/close_loop
//     PlcTask Inputs/MAIN.enable_stat[90] <-> Status process data mapping/enable
//     PlcTask Inputs/MAIN.force_rb_X[90] <-> Status process data mapping/force_rb_X
//     PlcTask Inputs/MAIN.force_rb_Y[90] <-> Status process data mapping/force_rb_Y
//     PlcTask Inputs/MAIN.force_rb_Z[90] <-> Status process data mapping/force_rb_Z
//     PlcTask Inputs/MAIN.force_sp_X[90] <-> Status process data mapping/force_sp_X
//     PlcTask Inputs/MAIN.force_sp_Y[90] <-> Status process data mapping/force_sp_Y
//     PlcTask Inputs/MAIN.force_sp_Z[90] <-> Status process data mapping/force_sp_Z
//     PlcTask Inputs/MAIN.pwm1[90] <-> Status process data mapping/pwm1
//     PlcTask Inputs/MAIN.pwm2[90] <-> Status process data mapping/pwm2
//     PlcTask Inputs/MAIN.pwm3[90] <-> Status process data mapping/pwm3
//     PlcTask Outputs/MAIN.enable_cmd[90] <-> Control process data mapping/enable
//     PlcTask Outputs/MAIN.force_cmd_X[90] <-> Control process data mapping/force_sp_X
//     PlcTask Outputs/MAIN.force_cmd_Y[90] <-> Control process data mapping/force_sp_Y
//     PlcTask Outputs/MAIN.force_cmd_Z[90] <-> Control process data mapping/force_sp_Z
//     PlcTask Outputs/MAIN.msthb[96] <-> Control process data mapping/msthb
//   SAsetGains/SAsetGains Instance <-> Device 1 (EtherCAT)/Box 97 (m1eph)
//     PlcTask Outputs/MAIN.msthb[97] <-> Control process data mapping/msthb
//   SAsetGains/SAsetGains Instance <-> Device 1 (EtherCAT)/Box 97 (m1eph)/Box 100 (m1sa)
//     PlcTask Inputs/MAIN.cloop_stat[93] <-> Status process data mapping/close_loop
//     PlcTask Inputs/MAIN.enable_stat[93] <-> Status process data mapping/enable
//     PlcTask Inputs/MAIN.force_rb_X[93] <-> Status process data mapping/force_rb_X
//     PlcTask Inputs/MAIN.force_rb_Y[93] <-> Status process data mapping/force_rb_Y
//     PlcTask Inputs/MAIN.force_rb_Z[93] <-> Status process data mapping/force_rb_Z
//     PlcTask Inputs/MAIN.force_sp_X[93] <-> Status process data mapping/force_sp_X
//     PlcTask Inputs/MAIN.force_sp_Y[93] <-> Status process data mapping/force_sp_Y
//     PlcTask Inputs/MAIN.force_sp_Z[93] <-> Status process data mapping/force_sp_Z
//     PlcTask Inputs/MAIN.pwm1[93] <-> Status process data mapping/pwm1
//     PlcTask Inputs/MAIN.pwm2[93] <-> Status process data mapping/pwm2
//     PlcTask Inputs/MAIN.pwm3[93] <-> Status process data mapping/pwm3
//     PlcTask Outputs/MAIN.enable_cmd[93] <-> Control process data mapping/enable
//     PlcTask Outputs/MAIN.force_cmd_X[93] <-> Control process data mapping/force_sp_X
//     PlcTask Outputs/MAIN.force_cmd_Y[93] <-> Control process data mapping/force_sp_Y
//     PlcTask Outputs/MAIN.force_cmd_Z[93] <-> Control process data mapping/force_sp_Z
//     PlcTask Outputs/MAIN.msthb[100] <-> Control process data mapping/msthb
//   SAsetGains/SAsetGains Instance <-> Device 1 (EtherCAT)/Box 97 (m1eph)/Box 101 (m1sa)
//     PlcTask Inputs/MAIN.cloop_stat[94] <-> Status process data mapping/close_loop
//     PlcTask Inputs/MAIN.enable_stat[94] <-> Status process data mapping/enable
//     PlcTask Inputs/MAIN.force_rb_X[94] <-> Status process data mapping/force_rb_X
//     PlcTask Inputs/MAIN.force_rb_Y[94] <-> Status process data mapping/force_rb_Y
//     PlcTask Inputs/MAIN.force_rb_Z[94] <-> Status process data mapping/force_rb_Z
//     PlcTask Inputs/MAIN.force_sp_X[94] <-> Status process data mapping/force_sp_X
//     PlcTask Inputs/MAIN.force_sp_Y[94] <-> Status process data mapping/force_sp_Y
//     PlcTask Inputs/MAIN.force_sp_Z[94] <-> Status process data mapping/force_sp_Z
//     PlcTask Inputs/MAIN.pwm1[94] <-> Status process data mapping/pwm1
//     PlcTask Inputs/MAIN.pwm2[94] <-> Status process data mapping/pwm2
//     PlcTask Inputs/MAIN.pwm3[94] <-> Status process data mapping/pwm3
//     PlcTask Outputs/MAIN.enable_cmd[94] <-> Control process data mapping/enable
//     PlcTask Outputs/MAIN.force_cmd_X[94] <-> Control process data mapping/force_sp_X
//     PlcTask Outputs/MAIN.force_cmd_Y[94] <-> Control process data mapping/force_sp_Y
//     PlcTask Outputs/MAIN.force_cmd_Z[94] <-> Control process data mapping/force_sp_Z
//     PlcTask Outputs/MAIN.msthb[101] <-> Control process data mapping/msthb
//   SAsetGains/SAsetGains Instance <-> Device 1 (EtherCAT)/Box 97 (m1eph)/Box 102 (m1sa)
//     PlcTask Inputs/MAIN.cloop_stat[95] <-> Status process data mapping/close_loop
//     PlcTask Inputs/MAIN.enable_stat[95] <-> Status process data mapping/enable
//     PlcTask Inputs/MAIN.force_rb_X[95] <-> Status process data mapping/force_rb_X
//     PlcTask Inputs/MAIN.force_rb_Y[95] <-> Status process data mapping/force_rb_Y
//     PlcTask Inputs/MAIN.force_rb_Z[95] <-> Status process data mapping/force_rb_Z
//     PlcTask Inputs/MAIN.force_sp_X[95] <-> Status process data mapping/force_sp_X
//     PlcTask Inputs/MAIN.force_sp_Y[95] <-> Status process data mapping/force_sp_Y
//     PlcTask Inputs/MAIN.force_sp_Z[95] <-> Status process data mapping/force_sp_Z
//     PlcTask Inputs/MAIN.pwm1[95] <-> Status process data mapping/pwm1
//     PlcTask Inputs/MAIN.pwm2[95] <-> Status process data mapping/pwm2
//     PlcTask Inputs/MAIN.pwm3[95] <-> Status process data mapping/pwm3
//     PlcTask Outputs/MAIN.enable_cmd[95] <-> Control process data mapping/enable
//     PlcTask Outputs/MAIN.force_cmd_X[95] <-> Control process data mapping/force_sp_X
//     PlcTask Outputs/MAIN.force_cmd_Y[95] <-> Control process data mapping/force_sp_Y
//     PlcTask Outputs/MAIN.force_cmd_Z[95] <-> Control process data mapping/force_sp_Z
//     PlcTask Outputs/MAIN.msthb[102] <-> Control process data mapping/msthb
//   SAsetGains/SAsetGains Instance <-> Device 1 (EtherCAT)/Box 97 (m1eph)/Box 103 (m1sa)
//     PlcTask Inputs/MAIN.cloop_stat[96] <-> Status process data mapping/close_loop
//     PlcTask Inputs/MAIN.enable_stat[96] <-> Status process data mapping/enable
//     PlcTask Inputs/MAIN.force_rb_X[96] <-> Status process data mapping/force_rb_X
//     PlcTask Inputs/MAIN.force_rb_Y[96] <-> Status process data mapping/force_rb_Y
//     PlcTask Inputs/MAIN.force_rb_Z[96] <-> Status process data mapping/force_rb_Z
//     PlcTask Inputs/MAIN.force_sp_X[96] <-> Status process data mapping/force_sp_X
//     PlcTask Inputs/MAIN.force_sp_Y[96] <-> Status process data mapping/force_sp_Y
//     PlcTask Inputs/MAIN.force_sp_Z[96] <-> Status process data mapping/force_sp_Z
//     PlcTask Inputs/MAIN.pwm1[96] <-> Status process data mapping/pwm1
//     PlcTask Inputs/MAIN.pwm2[96] <-> Status process data mapping/pwm2
//     PlcTask Inputs/MAIN.pwm3[96] <-> Status process data mapping/pwm3
//     PlcTask Outputs/MAIN.enable_cmd[96] <-> Control process data mapping/enable
//     PlcTask Outputs/MAIN.force_cmd_X[96] <-> Control process data mapping/force_sp_X
//     PlcTask Outputs/MAIN.force_cmd_Y[96] <-> Control process data mapping/force_sp_Y
//     PlcTask Outputs/MAIN.force_cmd_Z[96] <-> Control process data mapping/force_sp_Z
//     PlcTask Outputs/MAIN.msthb[103] <-> Control process data mapping/msthb
//   SAsetGains/SAsetGains Instance <-> Device 1 (EtherCAT)/Box 97 (m1eph)/Box 104 (m1sa)
//     PlcTask Inputs/MAIN.cloop_stat[97] <-> Status process data mapping/close_loop
//     PlcTask Inputs/MAIN.enable_stat[97] <-> Status process data mapping/enable
//     PlcTask Inputs/MAIN.force_rb_X[97] <-> Status process data mapping/force_rb_X
//     PlcTask Inputs/MAIN.force_rb_Y[97] <-> Status process data mapping/force_rb_Y
//     PlcTask Inputs/MAIN.force_rb_Z[97] <-> Status process data mapping/force_rb_Z
//     PlcTask Inputs/MAIN.force_sp_X[97] <-> Status process data mapping/force_sp_X
//     PlcTask Inputs/MAIN.force_sp_Y[97] <-> Status process data mapping/force_sp_Y
//     PlcTask Inputs/MAIN.force_sp_Z[97] <-> Status process data mapping/force_sp_Z
//     PlcTask Inputs/MAIN.pwm1[97] <-> Status process data mapping/pwm1
//     PlcTask Inputs/MAIN.pwm2[97] <-> Status process data mapping/pwm2
//     PlcTask Inputs/MAIN.pwm3[97] <-> Status process data mapping/pwm3
//     PlcTask Outputs/MAIN.enable_cmd[97] <-> Control process data mapping/enable
//     PlcTask Outputs/MAIN.force_cmd_X[97] <-> Control process data mapping/force_sp_X
//     PlcTask Outputs/MAIN.force_cmd_Y[97] <-> Control process data mapping/force_sp_Y
//     PlcTask Outputs/MAIN.force_cmd_Z[97] <-> Control process data mapping/force_sp_Z
//     PlcTask Outputs/MAIN.msthb[104] <-> Control process data mapping/msthb
//   SAsetGains/SAsetGains Instance <-> Device 1 (EtherCAT)/Box 97 (m1eph)/Box 105 (m1sa)
//     PlcTask Inputs/MAIN.cloop_stat[98] <-> Status process data mapping/close_loop
//     PlcTask Inputs/MAIN.enable_stat[98] <-> Status process data mapping/enable
//     PlcTask Inputs/MAIN.force_rb_X[98] <-> Status process data mapping/force_rb_X
//     PlcTask Inputs/MAIN.force_rb_Y[98] <-> Status process data mapping/force_rb_Y
//     PlcTask Inputs/MAIN.force_rb_Z[98] <-> Status process data mapping/force_rb_Z
//     PlcTask Inputs/MAIN.force_sp_X[98] <-> Status process data mapping/force_sp_X
//     PlcTask Inputs/MAIN.force_sp_Y[98] <-> Status process data mapping/force_sp_Y
//     PlcTask Inputs/MAIN.force_sp_Z[98] <-> Status process data mapping/force_sp_Z
//     PlcTask Inputs/MAIN.pwm1[98] <-> Status process data mapping/pwm1
//     PlcTask Inputs/MAIN.pwm2[98] <-> Status process data mapping/pwm2
//     PlcTask Inputs/MAIN.pwm3[98] <-> Status process data mapping/pwm3
//     PlcTask Outputs/MAIN.enable_cmd[98] <-> Control process data mapping/enable
//     PlcTask Outputs/MAIN.force_cmd_X[98] <-> Control process data mapping/force_sp_X
//     PlcTask Outputs/MAIN.force_cmd_Y[98] <-> Control process data mapping/force_sp_Y
//     PlcTask Outputs/MAIN.force_cmd_Z[98] <-> Control process data mapping/force_sp_Z
//     PlcTask Outputs/MAIN.msthb[105] <-> Control process data mapping/msthb
//   SAsetGains/SAsetGains Instance <-> Device 1 (EtherCAT)/Box 97 (m1eph)/Box 106 (m1sa)
//     PlcTask Inputs/MAIN.cloop_stat[99] <-> Status process data mapping/close_loop
//     PlcTask Inputs/MAIN.enable_stat[99] <-> Status process data mapping/enable
//     PlcTask Inputs/MAIN.force_rb_X[99] <-> Status process data mapping/force_rb_X
//     PlcTask Inputs/MAIN.force_rb_Y[99] <-> Status process data mapping/force_rb_Y
//     PlcTask Inputs/MAIN.force_rb_Z[99] <-> Status process data mapping/force_rb_Z
//     PlcTask Inputs/MAIN.force_sp_X[99] <-> Status process data mapping/force_sp_X
//     PlcTask Inputs/MAIN.force_sp_Y[99] <-> Status process data mapping/force_sp_Y
//     PlcTask Inputs/MAIN.force_sp_Z[99] <-> Status process data mapping/force_sp_Z
//     PlcTask Inputs/MAIN.pwm1[99] <-> Status process data mapping/pwm1
//     PlcTask Inputs/MAIN.pwm2[99] <-> Status process data mapping/pwm2
//     PlcTask Inputs/MAIN.pwm3[99] <-> Status process data mapping/pwm3
//     PlcTask Outputs/MAIN.enable_cmd[99] <-> Control process data mapping/enable
//     PlcTask Outputs/MAIN.force_cmd_X[99] <-> Control process data mapping/force_sp_X
//     PlcTask Outputs/MAIN.force_cmd_Y[99] <-> Control process data mapping/force_sp_Y
//     PlcTask Outputs/MAIN.force_cmd_Z[99] <-> Control process data mapping/force_sp_Z
//     PlcTask Outputs/MAIN.msthb[106] <-> Control process data mapping/msthb
//   SAsetGains/SAsetGains Instance <-> Device 1 (EtherCAT)/Box 97 (m1eph)/Box 107 (m1sa)
//     PlcTask Inputs/MAIN.cloop_stat[100] <-> Status process data mapping/close_loop
//     PlcTask Inputs/MAIN.enable_stat[100] <-> Status process data mapping/enable
//     PlcTask Inputs/MAIN.force_rb_X[100] <-> Status process data mapping/force_rb_X
//     PlcTask Inputs/MAIN.force_rb_Y[100] <-> Status process data mapping/force_rb_Y
//     PlcTask Inputs/MAIN.force_rb_Z[100] <-> Status process data mapping/force_rb_Z
//     PlcTask Inputs/MAIN.force_sp_X[100] <-> Status process data mapping/force_sp_X
//     PlcTask Inputs/MAIN.force_sp_Y[100] <-> Status process data mapping/force_sp_Y
//     PlcTask Inputs/MAIN.force_sp_Z[100] <-> Status process data mapping/force_sp_Z
//     PlcTask Inputs/MAIN.pwm1[100] <-> Status process data mapping/pwm1
//     PlcTask Inputs/MAIN.pwm2[100] <-> Status process data mapping/pwm2
//     PlcTask Inputs/MAIN.pwm3[100] <-> Status process data mapping/pwm3
//     PlcTask Outputs/MAIN.enable_cmd[100] <-> Control process data mapping/enable
//     PlcTask Outputs/MAIN.force_cmd_X[100] <-> Control process data mapping/force_sp_X
//     PlcTask Outputs/MAIN.force_cmd_Y[100] <-> Control process data mapping/force_sp_Y
//     PlcTask Outputs/MAIN.force_cmd_Z[100] <-> Control process data mapping/force_sp_Z
//     PlcTask Outputs/MAIN.msthb[107] <-> Control process data mapping/msthb
//   SAsetGains/SAsetGains Instance <-> Device 1 (EtherCAT)/Box 97 (m1eph)/Box 108 (m1sa)
//     PlcTask Inputs/MAIN.cloop_stat[101] <-> Status process data mapping/close_loop
//     PlcTask Inputs/MAIN.enable_stat[101] <-> Status process data mapping/enable
//     PlcTask Inputs/MAIN.force_rb_X[101] <-> Status process data mapping/force_rb_X
//     PlcTask Inputs/MAIN.force_rb_Y[101] <-> Status process data mapping/force_rb_Y
//     PlcTask Inputs/MAIN.force_rb_Z[101] <-> Status process data mapping/force_rb_Z
//     PlcTask Inputs/MAIN.force_sp_X[101] <-> Status process data mapping/force_sp_X
//     PlcTask Inputs/MAIN.force_sp_Y[101] <-> Status process data mapping/force_sp_Y
//     PlcTask Inputs/MAIN.force_sp_Z[101] <-> Status process data mapping/force_sp_Z
//     PlcTask Inputs/MAIN.pwm1[101] <-> Status process data mapping/pwm1
//     PlcTask Inputs/MAIN.pwm2[101] <-> Status process data mapping/pwm2
//     PlcTask Inputs/MAIN.pwm3[101] <-> Status process data mapping/pwm3
//     PlcTask Outputs/MAIN.enable_cmd[101] <-> Control process data mapping/enable
//     PlcTask Outputs/MAIN.force_cmd_X[101] <-> Control process data mapping/force_sp_X
//     PlcTask Outputs/MAIN.force_cmd_Y[101] <-> Control process data mapping/force_sp_Y
//     PlcTask Outputs/MAIN.force_cmd_Z[101] <-> Control process data mapping/force_sp_Z
//     PlcTask Outputs/MAIN.msthb[108] <-> Control process data mapping/msthb
//   SAsetGains/SAsetGains Instance <-> Device 1 (EtherCAT)/Box 97 (m1eph)/Box 109 (m1sa)
//     PlcTask Inputs/MAIN.cloop_stat[102] <-> Status process data mapping/close_loop
//     PlcTask Inputs/MAIN.enable_stat[102] <-> Status process data mapping/enable
//     PlcTask Inputs/MAIN.force_rb_X[102] <-> Status process data mapping/force_rb_X
//     PlcTask Inputs/MAIN.force_rb_Y[102] <-> Status process data mapping/force_rb_Y
//     PlcTask Inputs/MAIN.force_rb_Z[102] <-> Status process data mapping/force_rb_Z
//     PlcTask Inputs/MAIN.force_sp_X[102] <-> Status process data mapping/force_sp_X
//     PlcTask Inputs/MAIN.force_sp_Y[102] <-> Status process data mapping/force_sp_Y
//     PlcTask Inputs/MAIN.force_sp_Z[102] <-> Status process data mapping/force_sp_Z
//     PlcTask Inputs/MAIN.pwm1[102] <-> Status process data mapping/pwm1
//     PlcTask Inputs/MAIN.pwm2[102] <-> Status process data mapping/pwm2
//     PlcTask Inputs/MAIN.pwm3[102] <-> Status process data mapping/pwm3
//     PlcTask Outputs/MAIN.enable_cmd[102] <-> Control process data mapping/enable
//     PlcTask Outputs/MAIN.force_cmd_X[102] <-> Control process data mapping/force_sp_X
//     PlcTask Outputs/MAIN.force_cmd_Y[102] <-> Control process data mapping/force_sp_Y
//     PlcTask Outputs/MAIN.force_cmd_Z[102] <-> Control process data mapping/force_sp_Z
//     PlcTask Outputs/MAIN.msthb[109] <-> Control process data mapping/msthb
//   SAsetGains/SAsetGains Instance <-> Device 1 (EtherCAT)/Box 97 (m1eph)/Box 110 (m1sa)
//     PlcTask Inputs/MAIN.cloop_stat[103] <-> Status process data mapping/close_loop
//     PlcTask Inputs/MAIN.enable_stat[103] <-> Status process data mapping/enable
//     PlcTask Inputs/MAIN.force_rb_X[103] <-> Status process data mapping/force_rb_X
//     PlcTask Inputs/MAIN.force_rb_Y[103] <-> Status process data mapping/force_rb_Y
//     PlcTask Inputs/MAIN.force_rb_Z[103] <-> Status process data mapping/force_rb_Z
//     PlcTask Inputs/MAIN.force_sp_X[103] <-> Status process data mapping/force_sp_X
//     PlcTask Inputs/MAIN.force_sp_Y[103] <-> Status process data mapping/force_sp_Y
//     PlcTask Inputs/MAIN.force_sp_Z[103] <-> Status process data mapping/force_sp_Z
//     PlcTask Inputs/MAIN.pwm1[103] <-> Status process data mapping/pwm1
//     PlcTask Inputs/MAIN.pwm2[103] <-> Status process data mapping/pwm2
//     PlcTask Inputs/MAIN.pwm3[103] <-> Status process data mapping/pwm3
//     PlcTask Outputs/MAIN.enable_cmd[103] <-> Control process data mapping/enable
//     PlcTask Outputs/MAIN.force_cmd_X[103] <-> Control process data mapping/force_sp_X
//     PlcTask Outputs/MAIN.force_cmd_Y[103] <-> Control process data mapping/force_sp_Y
//     PlcTask Outputs/MAIN.force_cmd_Z[103] <-> Control process data mapping/force_sp_Z
//     PlcTask Outputs/MAIN.msthb[110] <-> Control process data mapping/msthb
//   SAsetGains/SAsetGains Instance <-> Device 1 (EtherCAT)/Box 97 (m1eph)/Box 111 (m1sa)
//     PlcTask Inputs/MAIN.cloop_stat[104] <-> Status process data mapping/close_loop
//     PlcTask Inputs/MAIN.enable_stat[104] <-> Status process data mapping/enable
//     PlcTask Inputs/MAIN.force_rb_X[104] <-> Status process data mapping/force_rb_X
//     PlcTask Inputs/MAIN.force_rb_Y[104] <-> Status process data mapping/force_rb_Y
//     PlcTask Inputs/MAIN.force_rb_Z[104] <-> Status process data mapping/force_rb_Z
//     PlcTask Inputs/MAIN.force_sp_X[104] <-> Status process data mapping/force_sp_X
//     PlcTask Inputs/MAIN.force_sp_Y[104] <-> Status process data mapping/force_sp_Y
//     PlcTask Inputs/MAIN.force_sp_Z[104] <-> Status process data mapping/force_sp_Z
//     PlcTask Inputs/MAIN.pwm1[104] <-> Status process data mapping/pwm1
//     PlcTask Inputs/MAIN.pwm2[104] <-> Status process data mapping/pwm2
//     PlcTask Inputs/MAIN.pwm3[104] <-> Status process data mapping/pwm3
//     PlcTask Outputs/MAIN.enable_cmd[104] <-> Control process data mapping/enable
//     PlcTask Outputs/MAIN.force_cmd_X[104] <-> Control process data mapping/force_sp_X
//     PlcTask Outputs/MAIN.force_cmd_Y[104] <-> Control process data mapping/force_sp_Y
//     PlcTask Outputs/MAIN.force_cmd_Z[104] <-> Control process data mapping/force_sp_Z
//     PlcTask Outputs/MAIN.msthb[111] <-> Control process data mapping/msthb
//   SAsetGains/SAsetGains Instance <-> Device 1 (EtherCAT)/Box 97 (m1eph)/Box 112 (m1sa)
//     PlcTask Inputs/MAIN.cloop_stat[105] <-> Status process data mapping/close_loop
//     PlcTask Inputs/MAIN.enable_stat[105] <-> Status process data mapping/enable
//     PlcTask Inputs/MAIN.force_rb_X[105] <-> Status process data mapping/force_rb_X
//     PlcTask Inputs/MAIN.force_rb_Y[105] <-> Status process data mapping/force_rb_Y
//     PlcTask Inputs/MAIN.force_rb_Z[105] <-> Status process data mapping/force_rb_Z
//     PlcTask Inputs/MAIN.force_sp_X[105] <-> Status process data mapping/force_sp_X
//     PlcTask Inputs/MAIN.force_sp_Y[105] <-> Status process data mapping/force_sp_Y
//     PlcTask Inputs/MAIN.force_sp_Z[105] <-> Status process data mapping/force_sp_Z
//     PlcTask Inputs/MAIN.pwm1[105] <-> Status process data mapping/pwm1
//     PlcTask Inputs/MAIN.pwm2[105] <-> Status process data mapping/pwm2
//     PlcTask Inputs/MAIN.pwm3[105] <-> Status process data mapping/pwm3
//     PlcTask Outputs/MAIN.enable_cmd[105] <-> Control process data mapping/enable
//     PlcTask Outputs/MAIN.force_cmd_X[105] <-> Control process data mapping/force_sp_X
//     PlcTask Outputs/MAIN.force_cmd_Y[105] <-> Control process data mapping/force_sp_Y
//     PlcTask Outputs/MAIN.force_cmd_Z[105] <-> Control process data mapping/force_sp_Z
//     PlcTask Outputs/MAIN.msthb[112] <-> Control process data mapping/msthb
//   SAsetGains/SAsetGains Instance <-> Device 1 (EtherCAT)/Box 97 (m1eph)/Box 113 (m1sa)
//     PlcTask Inputs/MAIN.cloop_stat[106] <-> Status process data mapping/close_loop
//     PlcTask Inputs/MAIN.enable_stat[106] <-> Status process data mapping/enable
//     PlcTask Inputs/MAIN.force_rb_X[106] <-> Status process data mapping/force_rb_X
//     PlcTask Inputs/MAIN.force_rb_Y[106] <-> Status process data mapping/force_rb_Y
//     PlcTask Inputs/MAIN.force_rb_Z[106] <-> Status process data mapping/force_rb_Z
//     PlcTask Inputs/MAIN.force_sp_X[106] <-> Status process data mapping/force_sp_X
//     PlcTask Inputs/MAIN.force_sp_Y[106] <-> Status process data mapping/force_sp_Y
//     PlcTask Inputs/MAIN.force_sp_Z[106] <-> Status process data mapping/force_sp_Z
//     PlcTask Inputs/MAIN.pwm1[106] <-> Status process data mapping/pwm1
//     PlcTask Inputs/MAIN.pwm2[106] <-> Status process data mapping/pwm2
//     PlcTask Inputs/MAIN.pwm3[106] <-> Status process data mapping/pwm3
//     PlcTask Outputs/MAIN.enable_cmd[106] <-> Control process data mapping/enable
//     PlcTask Outputs/MAIN.force_cmd_X[106] <-> Control process data mapping/force_sp_X
//     PlcTask Outputs/MAIN.force_cmd_Y[106] <-> Control process data mapping/force_sp_Y
//     PlcTask Outputs/MAIN.force_cmd_Z[106] <-> Control process data mapping/force_sp_Z
//     PlcTask Outputs/MAIN.msthb[113] <-> Control process data mapping/msthb
//   SAsetGains/SAsetGains Instance <-> Device 1 (EtherCAT)/Box 97 (m1eph)/Box 98 (m1sa)
//     PlcTask Inputs/MAIN.cloop_stat[91] <-> Status process data mapping/close_loop
//     PlcTask Inputs/MAIN.enable_stat[91] <-> Status process data mapping/enable
//     PlcTask Inputs/MAIN.force_rb_X[91] <-> Status process data mapping/force_rb_X
//     PlcTask Inputs/MAIN.force_rb_Y[91] <-> Status process data mapping/force_rb_Y
//     PlcTask Inputs/MAIN.force_rb_Z[91] <-> Status process data mapping/force_rb_Z
//     PlcTask Inputs/MAIN.force_sp_X[91] <-> Status process data mapping/force_sp_X
//     PlcTask Inputs/MAIN.force_sp_Y[91] <-> Status process data mapping/force_sp_Y
//     PlcTask Inputs/MAIN.force_sp_Z[91] <-> Status process data mapping/force_sp_Z
//     PlcTask Inputs/MAIN.pwm1[91] <-> Status process data mapping/pwm1
//     PlcTask Inputs/MAIN.pwm2[91] <-> Status process data mapping/pwm2
//     PlcTask Inputs/MAIN.pwm3[91] <-> Status process data mapping/pwm3
//     PlcTask Outputs/MAIN.enable_cmd[91] <-> Control process data mapping/enable
//     PlcTask Outputs/MAIN.force_cmd_X[91] <-> Control process data mapping/force_sp_X
//     PlcTask Outputs/MAIN.force_cmd_Y[91] <-> Control process data mapping/force_sp_Y
//     PlcTask Outputs/MAIN.force_cmd_Z[91] <-> Control process data mapping/force_sp_Z
//     PlcTask Outputs/MAIN.msthb[98] <-> Control process data mapping/msthb
//   SAsetGains/SAsetGains Instance <-> Device 1 (EtherCAT)/Box 97 (m1eph)/Box 99 (m1sa)
//     PlcTask Inputs/MAIN.cloop_stat[92] <-> Status process data mapping/close_loop
//     PlcTask Inputs/MAIN.enable_stat[92] <-> Status process data mapping/enable
//     PlcTask Inputs/MAIN.force_rb_X[92] <-> Status process data mapping/force_rb_X
//     PlcTask Inputs/MAIN.force_rb_Y[92] <-> Status process data mapping/force_rb_Y
//     PlcTask Inputs/MAIN.force_rb_Z[92] <-> Status process data mapping/force_rb_Z
//     PlcTask Inputs/MAIN.force_sp_X[92] <-> Status process data mapping/force_sp_X
//     PlcTask Inputs/MAIN.force_sp_Y[92] <-> Status process data mapping/force_sp_Y
//     PlcTask Inputs/MAIN.force_sp_Z[92] <-> Status process data mapping/force_sp_Z
//     PlcTask Inputs/MAIN.pwm1[92] <-> Status process data mapping/pwm1
//     PlcTask Inputs/MAIN.pwm2[92] <-> Status process data mapping/pwm2
//     PlcTask Inputs/MAIN.pwm3[92] <-> Status process data mapping/pwm3
//     PlcTask Outputs/MAIN.enable_cmd[92] <-> Control process data mapping/enable
//     PlcTask Outputs/MAIN.force_cmd_X[92] <-> Control process data mapping/force_sp_X
//     PlcTask Outputs/MAIN.force_cmd_Y[92] <-> Control process data mapping/force_sp_Y
//     PlcTask Outputs/MAIN.force_cmd_Z[92] <-> Control process data mapping/force_sp_Z
//     PlcTask Outputs/MAIN.msthb[99] <-> Control process data mapping/msthb

CONFIGURATION SAsetGains
    RESOURCE PLC ON TwinCAT3
        TASK PlcTask(INTERVAL := T#10ms, PRIORITY := 20);
        PROGRAM MAIN WITH PlcTask : MAIN;
        PROGRAM clear_fault WITH PlcTask : clear_fault;
        PROGRAM read_ncyl WITH PlcTask : read_ncyl;
        PROGRAM write_gains WITH PlcTask : write_gains;
        PROGRAM save_soc WITH PlcTask : save_soc;
        PROGRAM read_alias WITH PlcTask : read_alias;
        PROGRAM read_dongle WITH PlcTask : read_dongle;
    END_RESOURCE
END_CONFIGURATION

// ---- POUs/MAIN.TcPOU
PROGRAM MAIN
VAR
	// heartbeat
	msthb AT %Q* : ARRAY[1..181] OF UDINT;
	sa_indx : INT :=1;
	
	// enable, diable 
	enable_all : BOOL := FALSE;
	disable_all : BOOL := FALSE;
	enable_cmd AT %Q* : ARRAY[1..170] OF BOOL;
	cloop_stat AT %I* : ARRAY[1..170] OF BOOL;
	enable_stat AT %I* : ARRAY[1..170] OF BOOL;
	
	// clear fault
	slv_addr : UINT := 1002;
	clear_all : BOOL := FALSE;
	ctrl_clear_error :  BOOL;
	delay_cycle : UINT := 1;
	
	// bump test all SAa
	bump_start : BOOL := FALSE;
	bump_force : REAL := 0;
	bump_stop : BOOL := FALSE;
	bump_axis : INT := 1;
	delay_cycle2 : UINT := 1;
	sa_indx2 : INT :=1;
	
	// ramp signal test
	ramp_stop : BOOL;
	ramp_start: BOOL;
	ramp_start_single :BOOL;
	slope : REAL;
	ramp_cmd : REAL;	
	
	// read ncyl
	read_ncyl : BOOL;
	sa_indx3 : INT :=1;
	slv_addr_ncyl : UINT :=1002;
	
	// read alias
	read_alias : BOOL;
	sa_indx7 : INT :=1;
	slv_addr_alias : UINT :=1002;
	
	// read dongle
	read_dongle : BOOL;
	// sa_indx7 : INT :=1;
	slv_addr_dongle : UINT :=1002;
	dongle_nSubIndex : BYTE;
	Fx_min :ARRAY[1..170] OF REAL;
	Fy_min :ARRAY[1..170] OF REAL;
	Fz_min :ARRAY[1..170] OF REAL;
	Fx_max :ARRAY[1..170] OF REAL;
	Fy_max :ARRAY[1..170] OF REAL;	
	Fz_max :ARRAY[1..170] OF REAL;
	
	// write gains
	write_gains : BOOL ;
	write_SAgains : BOOL;
	slv_addr_ncyl2 : UINT :=1002;
	sa_indx4 : INT :=1;
	subindex: BYTE := 16#04;
	cylindex : WORD := 16#8001;
	kp : REAL :=1.2;
	ki : REAL := 0.8;
	kd : REAL := 0.0;
	dbp : REAL := 14;
	dbn : REAL := -14;
	dbi : REAL := 0.5;
	gval : REAL := kp;
	
	// save_soc
	slv_addr_soc : UINT := 1002;
	save_soc_all : BOOL := FALSE;
	delay_cycle4 : UINT := 1;
	
	// single SA Step
	set_zero: BOOL;
	singleSA_step: BOOL;
	force : REAL := 0.0;
	sa_indx5: INT := 1;
	axis: INT := 1;
	delay_cycle3: INT;
	sa_indx6: INT := 1;
	
	//Force vectors
	// control
	force_cmd_X AT %Q* : ARRAY[1..170] OF REAL;
	force_cmd_Y AT %Q* : ARRAY[1..170] OF REAL;
	force_cmd_Z AT %Q* : ARRAY[1..170] OF REAL;
	
	// status
	force_rb_X AT %I* : ARRAY[1..170] OF REAL;
	force_rb_Y AT %I* : ARRAY[1..170] OF REAL;
	force_rb_Z AT %I* : ARRAY[1..170] OF REAL;
	force_sp_X AT %I* : ARRAY[1..170] OF REAL;
	force_sp_Y AT %I* : ARRAY[1..170] OF REAL;
	force_sp_Z AT %I* : ARRAY[1..170] OF REAL;
	
	
	//pwm
	pwm1 AT %I* : ARRAY[1..170] OF REAL;
	pwm2 AT %I* : ARRAY[1..170] OF REAL;
	pwm3 AT %I* : ARRAY[1..170] OF REAL;
	
	// Network parameters
	sNetId_local : T_AmsNetId := '10.10.16.19.2.1';	// Address of this computer 
	FrmWcStat AT %I* : ARRAY[1..7] OF UINT;
	
	// scope vars
	scope_spX : REAL;
	scope_spY : REAL;
	scope_spZ : REAL;
	scope_rbX : REAL;
	scope_rbY : REAL;
	scope_rbZ : REAL;
	scope_pwm1 : REAL;
	scope_pwm2 : REAL;
	scope_pwm3 : REAL;
	scope_alias : UINT;
	scope_cyl :UDINT;


	c: INT :=0;
END_VAR

VAR_INPUT
	cyl : ARRAY[1..170] OF UDINT;
	alias : ARRAY[1..170] OF UINT;
	value : ARRAY[1..170] OF REAL;
END_VAR

// send heartbeat to all SA and EPHS
FOR sa_indx := 1 TO 181 BY 1 DO
	msthb[sa_indx] := msthb[sa_indx] + 1;
END_FOR


// clear fault on all SAs
IF (clear_all = TRUE AND slv_addr<1182) THEN
	ctrl_clear_error := TRUE;
	IF delay_cycle = 10 THEN
		slv_addr := slv_addr + 1;
		CASE  slv_addr OF
			1001,1018,1033,1046,1063,1080,1097,1114,1131,1148,1165:
			slv_addr := slv_addr+1;
		END_CASE
		delay_cycle := 1;
	ELSE
		delay_cycle := delay_cycle+1;	
	END_IF
	
ELSE
	slv_addr := 1002;
	ctrl_clear_error := FALSE;
END_IF

// send enable signal to all SAs
IF enable_all = TRUE THEN
	FOR sa_indx := 1 TO 170 BY 1 DO
		enable_cmd[sa_indx] := TRUE;
	END_FOR
END_IF

// send disable signal to all SAs
IF disable_all = TRUE THEN
	FOR sa_indx := 1 TO 170 BY 1 DO
		enable_cmd[sa_indx] := FALSE;
	END_FOR
	enable_all := FALSE;
END_IF

// Do xyz axis bump test on all SAs
IF bump_stop = TRUE THEN;
	bump_start := FALSE;
	sa_indx2 := 2;
	bump_axis := 0;
	delay_cycle2 := 0;
	FOR sa_indx := 1 TO 170 BY 1 DO
		force_cmd_X[sa_indx] := 0;
		force_cmd_Y[sa_indx] := 0; 
		force_cmd_Z[sa_indx] := 0;
		
	END_FOR
END_IF

IF bump_start = TRUE THEN
	IF delay_cycle2 = 500 THEN
		delay_cycle2 := 1;
		IF bump_axis < 3 THEN
			bump_axis := bump_axis +1;
		ELSE
			bump_axis := 1;
		END_IF
		IF bump_axis = 1 THEN
			sa_indx2 := sa_indx2 + 1;
			IF sa_indx2 > 170 THEN
				sa_indx2 := 2;
			END_IF
		END_IF
			
	ELSE
		delay_cycle2 := delay_cycle2+1;
		scope_spX := force_sp_x[sa_indx2];
		scope_spY := force_sp_y[sa_indx2];
		scope_spZ := force_sp_z[sa_indx2];
		scope_rbX := force_rb_x[sa_indx2];
		scope_rbY := force_rb_y[sa_indx2];
		scope_rbZ := force_rb_z[sa_indx2];
		scope_pwm1 := pwm1[sa_indx2];
		scope_pwm2 := pwm2[sa_indx2];
		scope_pwm3 := pwm3[sa_indx2];
		scope_alias := alias[sa_indx2];
		CASE bump_axis OF
			1 :
			force_cmd_X[sa_indx2] := bump_force;
			force_cmd_X[sa_indx2-1] := 0;
			force_cmd_Z[sa_indx2] := 0;
			2 :
			force_cmd_Y[sa_indx2] := bump_force;
			force_cmd_Y[sa_indx2-1] := 0;
			force_cmd_X[sa_indx2] := 0;
			3 :
			force_cmd_Z[sa_indx2] := bump_force;
			force_cmd_Z[sa_indx2-1] := 0;
			force_cmd_Y[sa_indx2] := 0;
		END_CASE
			
	END_IF
END_IF



// Do ramp test on all SAs
IF ramp_stop = TRUE THEN;
	ramp_start := FALSE;
	ramp_start_single := FALSE;
	ramp_cmd := 0.0;
	sa_indx2 := 1;
	bump_axis := 0;
	delay_cycle2 := 0;
	FOR sa_indx := 1 TO 170 BY 1 DO
		force_cmd_X[sa_indx] := 0;
		force_cmd_Y[sa_indx] := 0; 
		force_cmd_Z[sa_indx] := 0;
		
	END_FOR
END_IF

IF ramp_start = TRUE THEN
	ramp_start_single := FALSE;
	IF delay_cycle2 = 500 THEN
		delay_cycle2 := 1;
		slope := -slope;
		ramp_cmd := 0;
		IF cyl[sa_indx2] = 3 THEN
			IF bump_axis < 3 THEN
				bump_axis := bump_axis +1;
			ELSE
				bump_axis := 1;
			END_IF
		ELSE
			bump_axis := 1;
		END_IF		
	ELSE
		delay_cycle2 := delay_cycle2+1;
		scope_spX := force_sp_x[sa_indx2];
		scope_spY := force_sp_y[sa_indx2];
		scope_spZ := force_sp_z[sa_indx2];
		scope_rbX := force_rb_x[sa_indx2];
		scope_rbY := force_rb_y[sa_indx2];
		scope_rbZ := force_rb_z[sa_indx2];
		scope_pwm1 := pwm1[sa_indx2];
		scope_pwm2 := pwm2[sa_indx2];
		scope_pwm3 := pwm3[sa_indx2];
		scope_alias := alias[sa_indx2];
		scope_cyl := cyl[sa_indx2];
		
		IF ramp_cmd > 250*abs(slope) THEN
			slope := -1*slope;
		END_IF
		ramp_cmd := ramp_cmd + slope;
		CASE bump_axis OF
			1 :
			force_cmd_Z[sa_indx2] := ramp_cmd;
			IF sa_indx2 <> 1 THEN
				force_cmd_Y[sa_indx2-1] := 0;
				force_cmd_X[sa_indx2-1] := 0;	
			END_IF
		
			2 :
			force_cmd_Y[sa_indx2] := ramp_cmd;
			IF sa_indx2 <> 1 THEN
				force_cmd_X[sa_indx2-1] := 0;
				force_cmd_Z[sa_indx2] := 0;	
			END_IF
			3 :
			force_cmd_X[sa_indx2] := ramp_cmd;
			IF sa_indx2 <> 1 THEN
				force_cmd_Y[sa_indx2] := 0;
				force_cmd_Z[sa_indx2-1] := 0;	
			END_IF
		END_CASE	
	END_IF
	IF bump_axis = 1 AND delay_cycle2 =500  THEN
				sa_indx2 := sa_indx2 + 1;				
	END_IF
	IF sa_indx2 > 170 THEN
			sa_indx2 := 1;
	END_IF
END_IF

// ramp single axis

IF ramp_start_single = TRUE THEN
	ramp_start := FALSE;
	IF delay_cycle2 = 500 THEN
		delay_cycle2 := 1;
		slope := -slope;
		ramp_cmd := 0;
		IF cyl[sa_indx2] = 3 THEN
			IF bump_axis < 3 THEN
				bump_axis := bump_axis +1;
			ELSE
				bump_axis := 1;
			END_IF	
		ELSE
			bump_axis := 3;
		END_IF			
	ELSE
		delay_cycle2 := delay_cycle2+1;
		scope_spX := force_sp_x[sa_indx2];
		scope_spY := force_sp_y[sa_indx2];
		scope_spZ := force_sp_z[sa_indx2];
		scope_rbX := force_rb_x[sa_indx2];
		scope_rbY := force_rb_y[sa_indx2];
		scope_rbZ := force_rb_z[sa_indx2];
		scope_pwm1 := pwm1[sa_indx2];
		scope_pwm2 := pwm2[sa_indx2];
		scope_pwm3 := pwm3[sa_indx2];
		
		scope_alias := alias[sa_indx2];
		scope_cyl := cyl[sa_indx2];
		
		
		IF ramp_cmd > 250*abs(slope) THEN
			slope := -1*slope;
		END_IF
		ramp_cmd := ramp_cmd + slope;
		CASE bump_axis OF
			1 :
			force_cmd_X[sa_indx2] := ramp_cmd;
			2 :
			force_cmd_Y[sa_indx2] := ramp_cmd;
			3 :
			force_cmd_Z[sa_indx2] := ramp_cmd;
		END_CASE
			
	END_IF
END_IF

// read ncyls on all SAs
IF (read_ncyl = TRUE AND slv_addr_ncyl<1182) THEN
	IF delay_cycle = 10 THEN
		slv_addr_ncyl := slv_addr_ncyl + 1;
		CASE  slv_addr_ncyl OF
			1001,1018,1033,1046,1063,1080,1097,1114,1131,1148,1165:
			slv_addr_ncyl := slv_addr_ncyl+1;
		END_CASE
		sa_indx3 := sa_indx3 + 1;
		delay_cycle := 1;
	ELSE
		delay_cycle := delay_cycle+1;	
	END_IF
	
ELSE
	slv_addr_ncyl := 1002;
	//ctrl_clear_error := FALSE;
	sa_indx3 := 1;
END_IF



// read alias on all SAs
IF (read_alias = TRUE AND slv_addr_alias<1182) THEN
	IF delay_cycle = 10 THEN
		slv_addr_alias := slv_addr_alias + 1;
		CASE  slv_addr_alias OF
			1001,1018,1033,1046,1063,1080,1097,1114,1131,1148,1165:
			slv_addr_alias := slv_addr_alias+1;
		END_CASE
		sa_indx7 := sa_indx7 + 1;
		delay_cycle := 1;
	ELSE
		delay_cycle := delay_cycle+1;	
	END_IF
	
ELSE
	slv_addr_alias := 1002;
	//ctrl_clear_error := FALSE;
	sa_indx7 := 1;
END_IF

// read dongles on all SAs

//IF (read_dongle = TRUE AND slv_addr_dongle<1181) THEN
//	IF delay_cycle = 10 THEN
//		//dongle_nSubIndex :=16#03;
//		slv_addr_dongle := slv_addr_dongle + 1;
//		CASE  slv_addr_dongle OF
//			1001,1018,1033,1046,1063,1080,1097,1114,1131,1148,1165:
//			slv_addr_dongle := slv_addr_dongle+1;
//		END_CASE
//		sa_indx7 := sa_indx7 + 1;
//		delay_cycle := 1;
//	ELSE
//		delay_cycle := delay_cycle+1;	
//	END_IF
	
//ELSE
//	slv_addr_dongle := 1002;
//	//ctrl_clear_error := FALSE;
//	//sa_indx7 := 1;
//END_IF


// write gains
IF (write_gains = TRUE AND slv_addr_ncyl2<1181) THEN
	write_SAgains := FALSE;
	IF delay_cycle = 10 THEN
		slv_addr_ncyl2 := slv_addr_ncyl2 + 1;
		CASE  slv_addr_ncyl2 OF
			1001,1018,1033,1046,1063,1080,1097,1114,1131,1148,1165:
			slv_addr_ncyl2 := slv_addr_ncyl2+1;
		END_CASE
		sa_indx4 := sa_indx4 + 1;
		delay_cycle := 1;
	ELSE
		delay_cycle := delay_cycle+1;	
	END_IF	
ELSIF (write_gains = TRUE AND slv_addr_ncyl2 >= 1181) THEN
	slv_addr_ncyl2 := 1002;
	sa_indx4 := 1;
	CASE subindex OF
		16#04 :
			subindex := 16#05;
			gval := ki;
		16#05 :
			subindex := 16#0B;
			gval := dbp;
		16#0B :
			subindex := 16#0C;
		gval := dbn;
		16#0C :
			subindex := 16#0E;
			gval := dbi;
		16#0E :
			subindex := 16#04;
			gval := kp;
		ELSE
			subindex:= 16#04;
			gval :=kp;
	END_CASE
ELSE
	slv_addr_ncyl2 := 1002;
	sa_indx4 := 1;
END_IF


// save_soc
IF (save_soc_all = TRUE AND slv_addr_soc<1181) THEN
	IF delay_cycle4 = 10 THEN
		slv_addr_soc := slv_addr_soc + 1;
		CASE  slv_addr_soc OF
			1001,1018,1033,1046,1063,1080,1097,1114,1131,1148,1165:
			slv_addr_soc := slv_addr_soc+1;
		END_CASE
		delay_cycle4 := 1;
	ELSE
		delay_cycle4 := delay_cycle4+1;	
	END_IF
	
ELSE
	slv_addr_soc := 1002;
END_IF

// set 50 N step response for and actuator
// set zero to all actuators
IF set_zero = TRUE THEN
	FOR sa_indx6 := 1 TO 170 BY 1 DO 
		force_cmd_X[sa_indx6] := 0;
		force_cmd_Y[sa_indx6] := 0;
		force_cmd_Z[sa_indx6] := 0;
	END_FOR
END_IF

// Do single actuator set reposne
IF singleSA_step = TRUE THEN
	scope_spX := force_sp_x[sa_indx5];
	scope_spY := force_sp_y[sa_indx5];
	scope_spZ := force_sp_z[sa_indx5];
	scope_rbX := force_rb_x[sa_indx5];
	scope_rbY := force_rb_y[sa_indx5];
	scope_rbZ := force_rb_z[sa_indx5];
	scope_pwm1 := pwm1[sa_indx5];
	scope_pwm2 := pwm2[sa_indx5];
	scope_pwm3 := pwm3[sa_indx5];
	scope_alias := alias[sa_indx5];
	CASE axis OF 
		1:
		IF delay_cycle3 = 1000 THEN
			delay_cycle3 := 1;
			force_cmd_X[sa_indx5] := 0;	
			axis := 2;
		ELSE
			delay_cycle3 := delay_cycle3+1;
			force_cmd_X[sa_indx5] := force;	
		END_IF
		2:
		IF delay_cycle3 = 1000 THEN
			delay_cycle3 := 1;
			force_cmd_Y[sa_indx5] := 0;	
			axis := 3;
		ELSE
			delay_cycle3 := delay_cycle3+1;
			force_cmd_Y[sa_indx5] := force;	
		END_IF
		3:
		IF delay_cycle3 = 1000 THEN
			delay_cycle3 := 1;
			force_cmd_Z[sa_indx5] := 0;
			axis := 1;
		ELSE
			delay_cycle3 := delay_cycle3+1;
			force_cmd_Z[sa_indx5] := force;	
		END_IF
	END_CASE
ELSE
	axis := 1;
	delay_cycle3 := 1;
	force_cmd_X[sa_indx5] := 0;
	force_cmd_Y[sa_indx5] := 0;
	force_cmd_Z[sa_indx5] := 0;
	sa_indx5 := 1;
END_IF

// change gains of a single actuator
// write gains for slv_addr_ncyl2
IF (write_SAgains = TRUE) THEN
	write_gains := FALSE;
	IF delay_cycle = 10 THEN
	//	sa_indx4 := sa_indx4 + 1;
		delay_cycle := 1;
	ELSE
		delay_cycle := delay_cycle+1;	
		CASE subindex OF
			16#04 :
				subindex := 16#05;
				gval := ki;
			16#05 :
				subindex := 16#0B;
				gval := dbp;
			16#0B :
				subindex := 16#0C;
			gval := dbn;
			16#0C :
				subindex := 16#0E;
				gval := dbi;
			16#0E :
				subindex := 16#04;
				gval := kp;
			ELSE
				subindex:= 16#04;
				gval := kp;
		END_CASE
	END_IF
END_IF
	

// ramp single axis

END_PROGRAM

// ---- POUs/read_ncyl.TcPOU
PROGRAM read_ncyl
VAR
	fbSdoRead  : FB_EcCoESdoRead;
    //sNetId     : T_AmsNetId := '172.16.2.131.2.1';
    bExecute   : BOOL;
    nSlaveAddr : UINT := 1003;
    nIndex     : WORD := 16#8005;
    nSubIndex  : BYTE :=16#05;
    ncyl   : UDINT;
    bError     : BOOL;
    nErrId     : UDINT;
END_VAR


bExecute := MAIN.read_ncyl;
fbSdoRead(sNetId:= MAIN.sNetId_local,nSlaveAddr :=MAIN.slv_addr_ncyl, nIndex:=nIndex, nSubIndex :=nSubIndex, pDstBuf:= ADR(ncyl), cbBufLen:=SIZEOF(ncyl),bExecute:=bExecute);
MAIN.cyl[MAIN.sa_indx3] := ncyl;

IF NOT fbSdoRead.bBusy THEN
        bExecute := FALSE;
		//done	:= TRUE;
        IF NOT bError THEN 
                (* write successful *)
                bError := FALSE;
                nErrId := 0;
        ELSE 
                (* write failed *)
                bError := fbSdoRead.bError;
                nErrId := fbSdoRead.nErrId;
        END_IF
        fbSdoRead(bExecute := FALSE);
END_IF

END_PROGRAM

// ---- POUs/read_alias.TcPOU
PROGRAM read_alias
VAR
	fbSdoRead  : FB_EcCoESdoRead;
    //sNetId     : T_AmsNetId := '172.16.2.131.2.1';
    bExecute   : BOOL;
    nSlaveAddr : UINT := 1003;
    nIndex     : WORD := 16#8008;
    nSubIndex  : BYTE :=16#01;
    alias   : UINT;
    bError     : BOOL;
    nErrId     : UDINT;
END_VAR

bExecute := MAIN.read_alias;
fbSdoRead(sNetId:= MAIN.sNetId_local,nSlaveAddr :=MAIN.slv_addr_alias, nIndex:=nIndex, nSubIndex :=nSubIndex, pDstBuf:= ADR(alias), cbBufLen:=SIZEOF(alias),bExecute:=bExecute);
MAIN.alias[MAIN.sa_indx7] := alias;

IF NOT fbSdoRead.bBusy THEN
        bExecute := FALSE;
		//done	:= TRUE;
        IF NOT bError THEN 
                (* write successful *)
                bError := FALSE;
                nErrId := 0;
        ELSE 
                (* write failed *)
                bError := fbSdoRead.bError;
                nErrId := fbSdoRead.nErrId;
        END_IF
        fbSdoRead(bExecute := FALSE);
END_IF

END_PROGRAM

// ---- POUs/read_dongle.TcPOU
PROGRAM read_dongle
VAR
	fbSdoRead  : FB_EcCoESdoRead;
    //sNetId     : T_AmsNetId := '172.16.2.131.2.1';
    bExecute   : BOOL;
    nSlaveAddr : UINT := 1003;
    nIndex     : WORD := 16#8008;
    nSubIndex  : BYTE :=16#01;
    value1   : REAL;
    bError     : BOOL;
    nErrId     : UDINT;
END_VAR

bExecute := MAIN.read_dongle;
fbSdoRead(sNetId:= MAIN.sNetId_local,nSlaveAddr :=MAIN.slv_addr_dongle, nIndex:=nIndex, nSubIndex :=MAIN.dongle_nSubIndex, pDstBuf:= ADR(value1), cbBufLen:=SIZEOF(value1),bExecute:=bExecute);
MAIN.value[MAIN.sa_indx7] := value1;

IF NOT fbSdoRead.bBusy THEN
        bExecute := FALSE;
		//done	:= TRUE;
        IF NOT bError THEN 
                (* write successful *)
                bError := FALSE;
                nErrId := 0;
        ELSE 
                (* write failed *)
                bError := fbSdoRead.bError;
                nErrId := fbSdoRead.nErrId;
        END_IF
        fbSdoRead(bExecute := FALSE);
END_IF

END_PROGRAM

// ---- POUs/write_gains.TcPOU
PROGRAM write_gains
VAR
	fbSdoWrite      : FB_EcCoESdoWrite;
	nSlaveAddr      : UINT := 1003; (* Port Number of EtherCAT Slave *)
	Index_cyl1          : WORD := 16#8001; (* CoE Object Index *)
	//Index_cyl2          : WORD := 16#8002; (* CoE Object Index *)
	//Index_cyl3          : WORD := 16#8003; (* CoE Object Index *)
	SubIndex_kp       : BYTE := 16#04; (* Subindex of CoE Object *)
	SubIndex_ki       : BYTE := 16#05; (* Subindex of CoE Object *)
	SubIndex_dbp       : BYTE := 16#0B; (* Subindex of CoE Object *)
	SubIndex_dbn       : BYTE := 16#0C; (* Subindex of CoE Object *)
	SubIndex_dbi       : BYTE := 16#0E; (* Subindex of CoE Object *)
	ncyl 				: BYTE := 16#05;
	bExecute        : BOOL; (* rising edge starts writing to the CoE Object *)
	bError          : BOOL;
	nErrId          : UDINT;		
	clear_error: BOOL := TRUE;
	configured : BOOL := FALSE;
	done			: BOOL := FALSE;
	pAddr : INT := 1018;
	sNetId_local: INT;
END_VAR

bExecute := (MAIN.write_gains OR MAIN.write_SAgains);

fbSdoWrite(
        sNetId          := MAIN.sNetId_local,
        //nSlaveAddr      := nSlaveAddr,
		nSlaveAddr := MAIN.slv_addr_ncyl2,
        nIndex          := Main.cylindex,
        nSubIndex       := Main.subindex,
        pSrcBuf         := ADR(Main.gval),
        cbBufLen        := SIZEOF(Main.gval),
        bExecute        := bExecute
);

IF NOT fbSdoWrite.bBusy THEN
        bExecute := FALSE;
		//done	:= TRUE;
        IF NOT bError THEN 
                (* write successful *)
                bError := FALSE;
                nErrId := 0;
        ELSE 
                (* write failed *)
                bError := fbSdoWrite.bError;
                nErrId := fbSdoWrite.nErrId;
        END_IF
        fbSdoWrite(bExecute := FALSE);
END_IF

END_PROGRAM

// ---- POUs/clear_fault.TcPOU
PROGRAM clear_fault
VAR
	fbSdoWrite      : FB_EcCoESdoWrite;
	nSlaveAddr      : UINT := 1003; (* Port Number of EtherCAT Slave *)
	nIndex          : WORD := 16#8006; (* CoE Object Index *)
	nSubIndex       : BYTE := 16#01; (* Subindex of CoE Object *)
	bExecute        : BOOL; (* rising edge starts writing to the CoE Object *)
	bError          : BOOL;
	nErrId          : UDINT;		
	clear_error: BOOL := TRUE;
	configured : BOOL := FALSE;
	done			: BOOL := FALSE;
	pAddr : INT := 1018;
	sNetId_local: INT;
END_VAR

bExecute := MAIN.ctrl_clear_error;

fbSdoWrite(
        sNetId          := MAIN.sNetId_local,
        //nSlaveAddr      := nSlaveAddr,
		nSlaveAddr := MAIN.slv_addr,
        nIndex          := nIndex,
        nSubIndex       := nSubIndex,
        pSrcBuf         := ADR(clear_error),
        cbBufLen        := SIZEOF(clear_error),
        bExecute        := bExecute
);

IF NOT fbSdoWrite.bBusy THEN
        bExecute := FALSE;
		//done	:= TRUE;
        IF NOT bError THEN 
                (* write successful *)
                bError := FALSE;
                nErrId := 0;
        ELSE 
                (* write failed *)
                bError := fbSdoWrite.bError;
                nErrId := fbSdoWrite.nErrId;
        END_IF
        fbSdoWrite(bExecute := FALSE);
END_IF

END_PROGRAM

// ---- POUs/save_soc.TcPOU
PROGRAM save_soc
VAR
	fbSdoWrite      : FB_EcCoESdoWrite;
	//nSlaveAddr      : UINT := 1003; (* Port Number of EtherCAT Slave *)
	nIndex          : WORD := 16#8006; (* CoE Object Index *)
	nSubIndex       : BYTE := 16#02; (* Subindex of CoE Object *)
	bExecute        : BOOL; (* rising edge starts writing to the CoE Object *)
	bError          : BOOL;
	nErrId          : UDINT;		
	save_gains: BOOL := TRUE;
	configured : BOOL := FALSE;
	done			: BOOL := FALSE;
	pAddr : INT := 1018;
	sNetId_local: INT;
END_VAR

bExecute := MAIN.save_soc_all;

fbSdoWrite(
        sNetId          := MAIN.sNetId_local,
        //nSlaveAddr      := nSlaveAddr,
		nSlaveAddr := MAIN.slv_addr_soc,
        nIndex          := nIndex,
        nSubIndex       := nSubIndex,
        pSrcBuf         := ADR(save_gains),
        cbBufLen        := SIZEOF(save_gains),
        bExecute        := bExecute
);

IF NOT fbSdoWrite.bBusy THEN
        bExecute := FALSE;
		//done	:= TRUE;
        IF NOT bError THEN 
                (* write successful *)
                bError := FALSE;
                nErrId := 0;
        ELSE 
                (* write failed *)
                bError := fbSdoWrite.bError;
                nErrId := fbSdoWrite.nErrId;
        END_IF
        fbSdoWrite(bExecute := FALSE);
END_IF

END_PROGRAM

// ---- POUs/read_write_SA_gains.TcPOU
PROGRAM read_write_SA_gains
VAR
	fbSdoWrite      : FB_EcCoESdoWrite;
	fbSdoRead      : FB_EcCoESdoRead;
	nSlaveAddr      : UINT := 1003; (* Port Number of EtherCAT Slave *)
	Index_cyl1          : WORD := 16#8001; (* CoE Object Index *)
	Index_cyl2          : WORD := 16#8002; (* CoE Object Index *)
	Index_cyl3          : WORD := 16#8003; (* CoE Object Index *)
	Index_soc          : WORD := 16#8005; (* CoE Object Index *)
	SubIndex_kp       : BYTE := 16#04; (* Subindex of CoE Object *)
	SubIndex_ki       : BYTE := 16#05; (* Subindex of CoE Object *)
	SubIndex_dbp       : BYTE := 16#0B; (* Subindex of CoE Object *)
	SubIndex_dbn       : BYTE := 16#0C; (* Subindex of CoE Object *)
	SubIndex_dbi       : BYTE := 16#0E; (* Subindex of CoE Object *)
	ncyl 				: BYTE := 16#05;
	bExecute        : BOOL; (* rising edge starts writing to the CoE Object *)
	bError          : BOOL;
	nErrId          : UDINT;		
	clear_error: BOOL := TRUE;
	configured : BOOL := FALSE;
	done			: BOOL := FALSE;
	pAddr : INT := 1018;
	sNetId_local: INT;
END_VAR

END_PROGRAM
